// TwinCAT 3 PLC project bot53_plccode2
// ProgramVersion: 3.1.4022.7
// libraries:
//   CAA Memory, * (CAA Technical Workgroup)
//   Tc2_Math, * (Beckhoff Automation GmbH)
//   Tc2_SerialCom, * (Beckhoff Automation GmbH)
//   Tc2_Standard, * (Beckhoff Automation GmbH)
//   Tc2_System, * (Beckhoff Automation GmbH)
//   Tc2_Utilities, * (Beckhoff Automation GmbH)
//   Tc3_Database, * (Beckhoff Automation GmbH)
//   Tc3_IotBase, * (Beckhoff Automation GmbH)
//   Tc3_IotCommunicator, * (Beckhoff Automation GmbH)
//   Tc3_JsonXml, * (Beckhoff Automation GmbH)
//   Tc3_Module, * (Beckhoff Automation GmbH)
//   TcMatrix, * (Burks Engineering)
// project tree:
//   / CanRecTask.TcTTO, MqttTask.TcTTO, PlcTask.TcTTO
//   DUTs/ ST_IMU_STATE.TcDUT, ST_COMMAND.TcDUT, ST_FBDATA.TcDUT, ST_TARGETS.TcDUT, ST_UPCAM.TcDUT
//   GVLs/ GVL.TcGVL
//   POUs/ CanReceiver.TcPOU, constrain_angle.TcPOU, detectStabilizedAngle.TcPOU, DriveMotors.TcPOU, enable_disable_driver.TcPOU, FB_CanReceiver.TcPOU, FB_Mqtt.TcPOU, MAIN.TcPOU, motion_controller.TcPOU, MqttPrg.TcPOU, reset_errors.TcPOU, roundToTwoDecimalPlaces.TcPOU, set_encoder_odeometry.TcPOU, set_imu_odeometry.TcPOU, set_qr_info.TcPOU
//   POUs/kalman/ accum.TcPOU, angErrorCalc.TcPOU, angSpdCommandLimiter.TcPOU, angSpdCommandMixer.TcPOU, atan2.TcPOU, choldc1.TcPOU, choldcsl.TcPOU, cholsl.TcPOU, errorDegreeCalculator.TcPOU, forwardMovement.TcPOU, kalmanController.TcPOU, kalmanInit.TcPOU, kalmanStep.TcPOU, kinematicSolution.TcPOU, linPosErrGenerator.TcPOU, linSpdCommandLimiter.TcPOU, linSpdCommandMixer.TcPOU, localization.TcPOU, mulmat.TcPOU, myfmod.TcPOU, mySign.TcPOU, robotAutomation.TcPOU, setIdealAngle.TcPOU, ssub.TcPOU, sub_mat.TcPOU, transpose.TcPOU
// real-time tasks:
//   TASK CanRecTask: cycle T#2ms, priority 1, ADS port 350
//   TASK MqttTask: cycle T#10ms, priority 2, ADS port 351
//   TASK PlcTask: cycle T#2ms, priority 3, ADS port 352
// I/O:
//   DEVICE Device 3 (EtherCAT), AmsNetId 169.254.228.245.4.1
//     Term 1 (EK1960-2600) [EK1960-2600 TwinSAFE-Compact-Controller (4 x Relay, RJ45)]
//       modules: Module 1 (FSoE), Module 2 (FSOUT), Module 3 (FSLOGIC)
//       Term 2 (EL9410) [EL9410 E-Bus Power Supplier  (Diagnostics)]
//       Term 3 (EL3052) [EL3052 2Ch. Ana. Input 4-20mA]
//       Term 4 (EL2008-0015) [EL2008-0015 8Ch. Dig. Output 24V DC, 0.35A, not short-circuit proof]
//       Term 16 (EL9011) [EL9011 End Terminal]
//     Lifter_Driver [SOMANET CiA402 Drive]
//     Rotator_Driver [SOMANET CiA402 Drive]
//     Locomotion_R [SOMANET CiA402 Drive]
//     Locomotion_L [SOMANET CiA402 Drive]
//   DEVICE Device 1 (RT-Ethernet Adapter)
// variable links:
//   bot53_plccode2/bot53_plccode2 Instance <-> Device 3 (EtherCAT)/Lifter_Driver
//     MqttTask Inputs/GVL.robotdata.Position_Velocity.Lifter_position_actual_value <-> TxPDO Mapping 1/Position actual value
//     MqttTask Outputs/GVL.robotdata.Position_Velocity.Lifter_target_position <-> RxPDO Mapping 1/Target position
//     MqttTask Outputs/GVL.robotdata.motorCword[2] <-> RxPDO Mapping 1/Controlword
//     PlcTask Inputs/GVL.Lifter_modesOfOperationDisplay <-> TxPDO Mapping 1/Modes of operation display
//     PlcTask Inputs/GVL.Lifter_statusword <-> TxPDO Mapping 1/Statusword
//     PlcTask Inputs/GVL.batteryVoltageINT <-> TxPDO Mapping 1/batteryVoltage
//     PlcTask Inputs/GVL.robotdata.motorError[2] <-> TxPDO Mapping 1/Error code
//     PlcTask Outputs/GVL.Lifter_modesOfOperation <-> RxPDO Mapping 1/Modes of operation
//   bot53_plccode2/bot53_plccode2 Instance <-> Device 3 (EtherCAT)/Locomotion_L
//     MqttTask Outputs/GVL.robotdata.Position_Velocity.Locomotion_1_target_velocity <-> RxPDO Mapping 1/Target velocity
//     MqttTask Outputs/GVL.robotdata.motorCword[1] <-> RxPDO Mapping 1/Controlword
//     PlcTask Inputs/GVL.Locomotion_1_actual_pos <-> TxPDO Mapping 1/Position actual value
//     PlcTask Inputs/GVL.Locomotion_1_modesOfOperationDisplay <-> TxPDO Mapping 1/Modes of operation display
//     PlcTask Inputs/GVL.robotdata.Position_Velocity.Locomotion_1_actual_velocity <-> TxPDO Mapping 1/Velocity actual value
//     PlcTask Inputs/GVL.robotdata.motorError[1] <-> TxPDO Mapping 1/Error code
//     PlcTask Outputs/GVL.Locomotion_1_modesOfOperation <-> RxPDO Mapping 1/Modes of operation
//   bot53_plccode2/bot53_plccode2 Instance <-> Device 3 (EtherCAT)/Locomotion_R
//     MqttTask Outputs/GVL.robotdata.Position_Velocity.Locomotion_2_target_velocity <-> RxPDO Mapping 1/Target velocity
//     MqttTask Outputs/GVL.robotdata.motorCword[0] <-> RxPDO Mapping 1/Controlword
//     PlcTask Inputs/GVL.Locomotion_2_actual_pos <-> TxPDO Mapping 1/Position actual value
//     PlcTask Inputs/GVL.Locomotion_2_modesOfOperationDisplay <-> TxPDO Mapping 1/Modes of operation display
//     PlcTask Inputs/GVL.robotdata.Position_Velocity.Locomotion_2_actual_velocity <-> TxPDO Mapping 1/Velocity actual value
//     PlcTask Inputs/GVL.robotdata.motorError[0] <-> TxPDO Mapping 1/Error code
//     PlcTask Outputs/GVL.Locomotion_2_modesOfOperation <-> RxPDO Mapping 1/Modes of operation
//   bot53_plccode2/bot53_plccode2 Instance <-> Device 3 (EtherCAT)/Rotator_Driver
//     MqttTask Inputs/GVL.robotdata.Position_Velocity.Rotator_position_actual_value <-> TxPDO Mapping 1/Position actual value
//     MqttTask Outputs/GVL.robotdata.Position_Velocity.Rotator_target_position <-> RxPDO Mapping 1/Target position
//     MqttTask Outputs/GVL.robotdata.motorCword[3] <-> RxPDO Mapping 1/Controlword
//     PlcTask Inputs/GVL.Rotator_modesOfOperationDisplay <-> TxPDO Mapping 1/Modes of operation display
//     PlcTask Inputs/GVL.Rotator_statusword <-> TxPDO Mapping 1/Statusword
//     PlcTask Inputs/GVL.robotdata.motorError[3] <-> TxPDO Mapping 1/Error code
//     PlcTask Outputs/GVL.Rotator_modesOfOperation <-> RxPDO Mapping 1/Modes of operation
//   bot53_plccode2/bot53_plccode2 Instance <-> Device 3 (EtherCAT)/Term 1 (EK1960-2600)/Term 3 (EL3052)
//     PlcTask Inputs/GVL.robotdata.lifterDistance <-> AI Standard Channel 1/Value
//   bot53_plccode2/bot53_plccode2 Instance <-> Device 3 (EtherCAT)/Term 1 (EK1960-2600)/Term 4 (EL2008-0015)
//     MqttTask Outputs/GVL.robotdata.chargerContactor <-> Channel 3/Output
//     MqttTask Outputs/GVL.robotdata.driverContactor <-> Channel 1/Output
//     MqttTask Outputs/GVL.robotdata.pfEnableContactor <-> Channel 2/Output

CONFIGURATION bot53_plccode2
    RESOURCE PLC ON TwinCAT3
        TASK CanRecTask(INTERVAL := T#2ms, PRIORITY := 1);
        TASK MqttTask(INTERVAL := T#2ms, PRIORITY := 2);
        TASK PlcTask(INTERVAL := T#2ms, PRIORITY := 3);
        PROGRAM CanReceiver WITH CanRecTask : CanReceiver;
        PROGRAM MqttPrg WITH MqttTask : MqttPrg;
        PROGRAM robotAutomation WITH MqttTask : robotAutomation;
        PROGRAM MAIN WITH PlcTask : MAIN;
    END_RESOURCE
END_CONFIGURATION

// ---- DUTs/ST_IMU_STATE.TcDUT
TYPE ST_IMU_STATE :
STRUCT
	imu_x:LREAL;
	imu_y:LREAL;
	imu_euler:LREAL;
	acc_x:LREAL;
	gyro_z:LREAL;
	hr_acc_x:LREAL;
	hr_gyro_z:LREAL;
	timediff:LREAL;
	euler_yaw:LREAL;
END_STRUCT
END_TYPE

// ---- DUTs/ST_COMMAND.TcDUT
TYPE ST_COMMAND :
STRUCT
	command:INT;
	distance:LREAL;
	direction:INT;
	acc:LREAL;
	jerk:LREAL;
	spd:LREAL;
END_STRUCT
END_TYPE

// ---- DUTs/ST_FBDATA.TcDUT

TYPE ST_FBDATA :
STRUCT
    robot_x:LREAL;
	robot_y:LREAL;
	robot_yaw:LREAL;
	lifter:LREAL;
	rotator:LREAL;
	upcam_state:st_upcam;
	batteryStatus:BYTE;
	batteryVoltage :LREAL := 50;
	batteryRequestCurrent:LREAL;
	batterySOC:INT:=90;
	batteryCurrentCons:LREAL;
	batteryErrorFlag:INT;
	qr_tag:INT:=0;
	qr_x:INT;
	qr_y:INT;
	qr_angle:INT;
	qr_yaw:LREAL:=0;
	imu_state:ST_IMU_STATE;
	deviation_yaw:LREAL;
	deviation_y:LREAL;
	imu_r:LREAL;
	imu_omega:LREAL;
	imu_readtime:LREAL;
	encoder_x:LREAL;
	encoder_y:LREAL;
	encoder_yaw:LREAL;
	encoder_v:LREAL;
	robot_direction:BYTE:=0;
	motion_status :BYTE:=1;
	activeState:BYTE:=1;
	
	motorError AT%I*:ARRAY[0..3] OF INT;
	Jerk:LREAL:=JERK_LIMIT;
	Acc:LREAL:=ACCELERATION_LIMIT;
	Speed:LREAL:=SPEED_LIMIT;
	controller:INT;
	motorCword AT%Q*: ARRAY[0..3] OF INT;
	yaw_error:LREAL;
	encoder_omega:LREAL;
	encoder_slave0_speed:LREAL;
	encoder_slave1_speed:LREAL;
	encoderx_rel:LREAL;
	encodery_rel:LREAL;
	imux_rel:LREAL;
	imuy_rel:LREAL;
	wc1:LREAL;
	wc2:LREAL;
	driverContactor                            AT%Q* : BOOL := TRUE;
    pfEnableContactor                        AT%Q* : BOOL := TRUE;
    chargerContactor                        AT%Q* : BOOL := FALSE;
	lifterDistance AT%I* : INT := INT#0;
	Position_Velocity:ST_TARGETS;
	activecommand:INT;
	Locomotion_1_modesOfOperationDisplay    AT%I* : SINT;
	Locomotion_2_modesOfOperationDisplay    AT%I* : SINT;
    Rotator_modesOfOperationDisplay         AT%I* : SINT;
    Lifter_modesOfOperationDisplay          AT%I* : SINT;
  
	END_STRUCT
	END_TYPE

// ---- DUTs/ST_TARGETS.TcDUT
TYPE ST_TARGETS :
STRUCT
	Locomotion_1_target_velocity			AT%Q* : DINT;
	Locomotion_2_target_velocity 			AT%Q* : DINT;
	Locomotion_1_actual_velocity			AT%I* : DINT;
	Locomotion_2_actual_velocity 			AT%I* : DINT;
	Lifter_position_actual_value             AT%I* : DINT;
	Lifter_target_position                     AT%Q* : DINT;
	Rotator_target_position                 AT%Q* : DINT;
	Rotator_position_actual_value             AT%I* : DINT;
	Rotator_target_velocity                 AT%Q* : DINT;
	Rotator_actual_velocity             AT%I* : DINT;
END_STRUCT
END_TYPE

// ---- DUTs/ST_UPCAM.TcDUT
TYPE ST_UPCAM :
STRUCT
	up_camera_x:LREAL;
	up_camera_y:LREAL;
	up_camera_yaw:LREAL;
	up_camera_tag:STRING[10];
END_STRUCT
END_TYPE

// ---- GVLs/GVL.TcGVL
//{attribute 'qualified_only'}
VAR_GLOBAL CONSTANT
COMMAND_LOCOMOTION_DISABLE:BYTE:=BYTE#2;
COMMAND_LOCOMOTION_ENABLE:BYTE:=BYTE#14;
COMMAND_LIFTER_DISABLE:BYTE:=BYTE#6;
COMMAND_LIFTER_ENABLE:BYTE:=BYTE#7;
COMMAND_ROTATOR_DISABLE:BYTE:=BYTE#8;
COMMAND_ROTATOR_ENABLE:BYTE:=BYTE#9;
COMMAND_PF_ENADIS:BYTE:=BYTE#11;
COMMAND_DRIVER_ENADIS:BYTE:=BYTE#12;
COMMAND_RESET_ERRORS:BYTE:=BYTE#1;
COMMAND_SET_MOTIONLIMITS:BYTE:=BYTE#21;
COMMAND_TOGGLE_CONT:BYTE:=BYTE#33;
COMMAND_CANCEL_COMMAND:BYTE:=BYTE#36;
COMMAND_ANG_CORR:BYTE:=BYTE#32;
COMMAND_X_CORR:BYTE:=BYTE#34;
MOTION_ONGOING:BYTE:=BYTE#0;
GRID_DIM:INT:=INT#1;
//QR_TX_INTERVAL:LREAL:=LREAL#25;
MOTION_ENDED:BYTE:=BYTE#1;
MOTION_INFINITE:BYTE:=BYTE#2;
MOTION_HOLDED:BYTE:=BYTE#3;
MOTION_ANGLE:BYTE:=BYTE#4;
MOTION_LIFTER:BYTE:=BYTE#5;
STARTSTOP_CHARGE:BYTE:=BYTE#45;
MOTION_OBSTACLE:BYTE:=BYTE#7;
MOTION_ROTATE:BYTE:=BYTE#8;
CHARGING:BYTE:=BYTE#9;
LIFTER_UP_LIMIT:INT:=INT#14879;
LIFTER_DOWN_LIMIT:INT:=INT#32000;
LIFTER_UP:INT:=INT#16000;
LIFTER_DOWN:INT:=INT#25000;

MOTION_BRAKE:BYTE:=BYTE#10;
IMU_RESET :BYTE:=BYTE#11;
ANGLE_CORRECT:BYTE:=BYTE#12;
LOCATION_CORRECT:BYTE:=BYTE#13;
INIT:BYTE:=BYTE#14;
LIFTING_DONE:BYTE:=BYTE#15;
POD_ANGLE_CORRECT:BYTE:=BYTE#16;
ENC_RESET :BYTE:=BYTE#17;
PDO_CHARGE_OPENCLOSE:BYTE:=BYTE#18;
STOP_ON_QR :BYTE:=BYTE#19;
UPCAM_READ:BYTE:=BYTE#20;
ANGLE_CORR_ENDED :BYTE:=BYTE#50;
X_CORR_ENDED :BYTE:=BYTE#51;
POD_CORR_ENDED:BYTE:=BYTE#52;
IMU_RST_ENDED:BYTE:=BYTE#53;
CONT_TOGGLE_ENDED :BYTE:=BYTE#54;
MOVE_ENDED :BYTE:=BYTE#55;
TURN_ENDED :BYTE:=BYTE#56;
LIFT_ENDED :BYTE:=BYTE#57;
ROTATE_ENDED :BYTE:=BYTE#58;
SETLIMITS_ENDED :BYTE:=BYTE#59;
CHARGE_ENDED:BYTE:=BYTE#60;
UPCAM_READ_ENDED :BYTE:=BYTE#61;
LIFT_UP:BYTE:=BYTE#62;
LIFT_DOWN:BYTE:=BYTE#63;
LOST:BYTE:=BYTE#100;
MOTOR_ERROR:BYTE:=BYTE#105;
PLC_ERROR:BYTE:=BYTE#106;
IMU_ERROR:BYTE:=BYTE#107;
NO_QR_TIMEOUT:DINT:=DINT#50000000;
NO_ADS_TIMEOUT:DINT:=DINT#150;
QRCAM_ERROR:BYTE:=BYTE#110;
COMM_PROB:BYTE:=BYTE#111;
CMD_TIMEOUT :BYTE:=BYTE#112;
STOPPER_DOWN:BYTE:=BYTE#114;
UPCAM_ERROR:BYTE:=BYTE#115; //error states starting from 100
PLC_COMM_ERROR :BYTE:=BYTE#116;
BMS_ERROR:BYTE:=BYTE#120;
PDO_CHARGER_ERROR :BYTE:=BYTE#121;
CRI_BATT:BYTE:=BYTE#125;
OVER_CURR:BYTE:=BYTE#126;
CHARGE_ERROR:BYTE:=BYTE#127;
LOW_BATT:BYTE:=BYTE#130;
MOTOR_OVER_TEMP:BYTE:=BYTE#135;
BATT_ERROR:BYTE:=BYTE#150;
LIFTER_STATE_INCORRECT:BYTE:=BYTE#160;

 

SUCCESS:INT:=INT#0;
FAILURE:INT:=INT#2;
NEGATIVE_FAILURE:INT:=INT#3;
NULL_POINTER:INT:=INT#4;
ROBOT_RADIUS:LREAL:=LREAL#0.32;
WHEEL_RADIUS:LREAL:=LREAL#0.08;
REDUCER_RATIO:LREAL:=LREAL#12;
ROTATOR_RADIUS:LREAL:=LREAL#0.466;
TURN_JERK_LIMIT:LREAL:=LREAL#0.4;
TURN_ACCELERATION_LIMIT:LREAL:=LREAL#0.2;
TURN_VELOCITY_LIMIT:LREAL:=LREAL#0.2;


DECELERATION_LIMIT:LREAL:=LREAL#1;

PLC_CYCLE:LREAL:=LREAL#0.002;
ROTATOR_REDUCER_RATIO:LREAL:=LREAL#14;
ROTATOR_GEAR_RATIO:LREAL:=LREAL#7.6;
ROTRAD2DEC:LREAL:=(10000.0 * (ROTATOR_REDUCER_RATIO) * (ROTATOR_GEAR_RATIO) / (2.0 * PI));
DEC2R:LREAL:=LREAL#1/ROTRAD2DEC;
M2DEC:LREAL:=((10000.0 * (REDUCER_RATIO)) / (2.0 * PI * (WHEEL_RADIUS)));
DEC2M:LREAL:= (1.0 / (M2DEC));
MSN2RPM:LREAL:= ((((REDUCER_RATIO) * 1.0 * 60.0) / (2.0 * PI * (WHEEL_RADIUS))));
RPM2MSN:LREAL:=1/MSN2RPM;
OMEGA_DIFF_MAX:LREAL:= ((1.5 * 1.5) / (ROBOT_RADIUS * ROBOT_RADIUS) * (PLC_CYCLE));

END_VAR
VAR_GLOBAL
imu_euler_prev:LREAL;
qr_xstate:LREAL;
qr_ystate:LREAL;
slave0_speed:LREAL;
slave1_speed:LREAL;
ACCELERATION_LIMIT:LREAL:=LREAL#1;
JERK_LIMIT:LREAL:=LREAL#0.8;
SPEED_LIMIT:LREAL:=LREAL#1.5;
//******************KALMAN VARIABLES**********************************************
	LINSPDRATELIMIT:LREAL:= 0.7;
	LINPOS_Kp :LREAL:=0.85;
	TURNANG_Kp:LREAL:= 1.5;
	TURNFWD_Kp:LREAL:= 1.5;
	FORWARD_MAX_SPEED :LREAL:=1.5;
	LINJERKLIMIT:LREAL:= 20;
	ANGSPDRATELIMIT :INT:= 20;
	calibrationCount:INT:=0;
	gyroZmean:LREAL:=0;
	accXmean:LREAL:=0; 
	PosFdbckX,PosFdbckX_Rel:LREAL:=0;
	PosFdbckY,PosFdbckY_Rel:LREAL:=0;
	ThetaFdbck:LREAL:=0;
	xStart:LREAL:=0;
	yStart:LREAL:=0;
	xGoal:LREAL:=0;
	yGoal:LREAL:=0;
	idealAngle:LREAL:=0;
	AngPosCommand:LREAL:=0;
	robotAngle:LREAL:=0;
	linPosErr:LREAL:=0;
	kalLinSpd:LREAL:=0;
	kalAngSpd:LREAL:=0;
	linSpdCommandShaped:LREAL:=0;angSpdCommandShaped:LREAL:=0;angPosFdbckRobot_Abs:LREAL:=0;angPosFdbckRobot:LREAL:=0; angSpdFdbckRobot_:LREAL:=0; linPosFdbckRobot_x:LREAL:=0; linSpdFdbckRobot_x_:LREAL:=0;linSpdFdbckRobot:LREAL:=0;
	angSpdFdbckRobot:LREAL:=0; linPosFdbckRobot_y:LREAL:=0; linSpdFdbckRobot_y_:LREAL:=0;rightWheelFdbck:LREAL:=0;leftWheelFdbck:LREAL:=0;
	robot_state:BYTE:=0;modeEnable:BYTE:=0;missionCompleted:INT:=1;userCommand:BYTE:=0; readyFlag:BYTE:=0;
	rightMotorSpeedCommand:DINT;leftMotorSpeedCommand:DINT;
	posTheta_wrt_robot_enc:LREAL;
	forwardCommand:LREAL:= 0;
	accLimited :LREAL:= 0;
	LinSpdFdbck:LREAL:=0;accFdbck:LREAL:=0;linSpd:LREAL:=0;
	Id:DynamicMatrix;
	I:ARRAY[0..2,0..2] OF LREAL:=[1,0,0,0,1,0,0,0,1];
	F_kalman1:ARRAY[0..2,0..2] OF LREAL:=[1,0.002,0.000002,0,1,0.002,0,0,1];	
	Q_kalman1:ARRAY[0..2,0..2] OF LREAL:=[0,0,0,0,0,0,0,0,10];
	R_kalman1:ARRAY[0..1,0..1] OF LREAL:=[1,0,0,1000];
	x_kalman1:ARRAY[0..2,0..0] OF LREAL:=[0,0,0];
	P_kalman1:ARRAY[0..2,0..2]OF LREAL:=[1,0,0,0,1,0,0,0,1];
	z_kalman1:ARRAY[0..1,0..0] OF LREAL;
	K_kalman1:ARRAY[0..2,0..1]OF LREAL;
	H_kalman1:ARRAY[0..1,0..2] OF LREAL:=[1,0,0,0,1,0];
	F_kalman2:ARRAY[0..2,0..2] OF LREAL:=[1,0.002,0.000002,0,1,0.002,0,0,1];
	Q_kalman2:ARRAY[0..2,0..2] OF LREAL:=[0,0,0,0,0,0,0,0,10];
	R_kalman2:ARRAY[0..1,0..1] OF LREAL:=[1,0,0,1];
	x_kalman2:ARRAY[0..2,0..0] OF LREAL:=[0,0,0];
	P_kalman2:ARRAY[0..2,0..2] OF LREAL:=[1,0,0,0,1,0,0,0,10];
	z_kalman2:ARRAY[0..1,0..0] OF LREAL;
	K_kalman2:ARRAY[0..2,0..1]  OF LREAL;
	H_kalman2:ARRAY[0..1,0..2] OF LREAL:=[1,0,0,0,1,0];
	err_kalman2:ARRAY[0..1,0..0] OF LREAL;
	F_kalman3:ARRAY[0..2,0..2] OF LREAL:=[1,0,0,0,1,0,0,0,1];
	Q_kalman3:ARRAY[0..2,0..2]  OF LREAL:=[10,0,0,0,10,0,0,0,0.2];
	R_kalman3:ARRAY[0..2,0..2] OF LREAL:=[0.01,0,0,0,0.01,0,0,0,500]; 
	x_kalman3:ARRAY[0..2,0..0]OF LREAL:=[0,0,0];
	z_kalman3:ARRAY[0..2,0..0]OF LREAL:=[0,0,0];
	P_kalman3:ARRAY[0..2,0..2]OF  LREAL:=[1,0,0,0,1,0,0,0,1];
	H_kalman3:ARRAY[0..2,0..2] OF LREAL;
	K_kalman3:ARRAY[0..2,0..2]OF LREAL;
	theta_pos:LREAL := 0;
	kalman12_x:LREAL;
	kalman12_y :LREAL;
	err_kalman3:ARRAY[0..2,0..0]OF LREAL;

//******************KALMAN VARIABLES**********************************************

	CONTROLLER_TYPE:BYTE:=0;
	KALMAN_INITIALIZED:BOOL:=FALSE;
	Y_DEV_THRESHOLD:LREAL:=0.005;
	PF_OFFSET:LREAL:=-0.4;
	pf_valid:BYTE:=0;
	AWAY_COEFF:LREAL:=LREAL#1;
	TOWARDS_COEFF:LREAL:=LREAL#1;
    current_yaw_deg:LREAL;
    ads_lasttime:ULINT;
    lateral_direction_sign:INT;
	batteryVoltageINT  AT%I*:UDINT;
    away:LREAL;
	cancelcommand:BOOL;
	raw_qr_tag:INT;
      stabilization_yaw_deg:LREAL;
    winnerEvaluated:BOOL:=FALSE;
    imuXwins:BOOL:=FALSE;
	imuAngwins:BOOL:=FALSE;
    lastqrtime:ULINT;
	lastqrtagtime:ULINT;
    controller_coeff:LREAL;
    imuYwins:BOOL:=FALSE;
    encoderx_rel:LREAL;
    encodery_rel:LREAL;
    imux_rel:LREAL;
    imuy_rel:LREAL;
	grid_x:LREAL;
	grid_y:LREAL;
    local_x_before_motion:LREAL:=0;
     robotdata:ST_FBDATA;
    st_command:ST_COMMAND;
    command:ARRAY[0..5] OF LREAL;
    motion_index :DINT;
    max_location :DINT;
    motion_left  :ARRAY[0..299999] OF DINT;
	motion_lift  :ARRAY[0..299999] OF DINT;
	motion_rotator  :ARRAY[0..299999] OF DINT;
    motion_right :ARRAY[0..299999] OF DINT;
    motion_vel :ARRAY[0..299999] OF LREAL;
    motion  :ARRAY[0..299999] OF DINT;
    deviation_y:LREAL;
    deviation_yaw:LREAL;
    KpY:LREAL:=95;
    KpTht:LREAL:=0.03;
    //Locomotion_1
    Locomotion_1_modesOfOperation             AT%Q* : SINT := SINT#9;
    Locomotion_1_error_state_1                 AT%I* : UINT;
    Locomotion_1_error_state_2                 AT%I* : UINT;
    Locomotion_1_statusword                 AT%I* : UINT;
	Locomotion_1_actual_pos                 AT%I* : DINT;
    Locomotion_1_modesOfOperationDisplay     AT%I* : SINT;
    //Locomotion_2

    Locomotion_2_modesOfOperation             AT%Q* : SINT := SINT#9;
    Locomotion_2_error_state_1                 AT%I* : UINT;
    Locomotion_2_error_state_2                 AT%I* : UINT;
    Locomotion_2_statusword                 AT%I* : UINT;
    Locomotion_2_modesOfOperationDisplay     AT%I* : SINT;
	Locomotion_2_actual_pos                 AT%I* : DINT;
    //Rotator
   
    Rotator_modesOfOperation                 AT%Q* : SINT := SINT#8;
  
    Rotator_error_state_1                     AT%I* : UINT;
    Rotator_error_state_2                     AT%I* : UINT;
    Rotator_statusword                         AT%I* : UINT;
    Rotator_modesOfOperationDisplay         AT%I* : SINT;
    //Lifter
  
    Lifter_modesOfOperation                 AT%Q* : SINT := SINT#8;
   
    Lifter_error_state_1                     AT%I* : UINT;
    Lifter_error_state_2                     AT%I* : UINT;
    Lifter_statusword                         AT%I* : UINT;
    Lifter_modesOfOperationDisplay             AT%I* : SINT;
    receivedBytes :STRING;
    sendReceiveTrigger : BOOL;

    MQTT_ConnState:ETcIotMqttClientState;
    MQTT_Command:FB_IoTCommand;

    //Enable Signals for to be switched subsystems
   

 


END_VAR

// ---- POUs/CanReceiver.TcPOU
PROGRAM CanReceiver
VAR
	fbUdp1 : FB_CanReceiver;
END_VAR

fbUdp1();

END_PROGRAM

// ---- POUs/FB_CanReceiver.TcPOU
{attribute 'c++_compatible'}
FUNCTION_BLOCK FB_CanReceiver IMPLEMENTS ITcIoUdpProtocolRecv
VAR_INPUT
END_VAR
VAR_OUTPUT
END_VAR
VAR
	{attribute 'TcInitSymbol'}
	oid : OTCID; 
	ipUdp : ITcIoUdpProtocol;
	nUdpPort : UINT := 4444;
	nReceivedPakets : UINT;
	
	hrInit : HRESULT;
	hrSend  : HRESULT;  
END_VAR

IF ipUdp <> 0 THEN
	ipUdp.CheckReceived();
END_IF

{attribute 'conditionalshow'}
METHOD FB_exit : BOOL
VAR_INPUT
	bInCopyCode : BOOL; // if TRUE, the exit method is called for exiting an instance that is copied afterwards (online change).
END_VAR
IF NOT bInCopyCode THEN // no online change
	IF ipUdp <> 0 THEN 
		ipUdp.UnregisterReceiver(nUdpPort); // Shutdown
		FW_SafeRelease(ADR(ipUdp));
		FB_exit := TRUE; 
	END_IF
END_IF
END_METHOD

{attribute 'conditionalshow'}
METHOD FB_init : BOOL
VAR_INPUT
	bInitRetains : BOOL; // if TRUE, the retain variables are initialized (warm start / cold start)
	bInCopyCode : BOOL;  // if TRUE, the instance afterwards gets moved into the copy code (online change)
END_VAR
VAR
	ipSrv : ITComObjectServer;

END_VAR
IF NOT bInCopyCode THEN // no online change
	IF ipUdp = 0 AND oid <> 0 THEN
	    hrInit := FW_ObjMgr_GetObjectInstance(	oid:=oid, 
											iid:=TC_GLOBAL_IID_LIST.IID_ITcIoUdpProtocol, 
											pipUnk:=ADR(ipUdp) );
		IF SUCCEEDED(hrInit) THEN 
			IF  SUCCEEDED(ipUdp.RegisterReceiver(nUdpPort, THIS^)) THEN //open port
				FB_init := TRUE;
			ELSE 
				FB_init := FALSE; 
				FW_SafeRelease(ADR(ipUdp));
			END_IF
		END_IF
	ELSIF oid = 0 THEN 
		FB_init := FALSE; 
		hrInit := ERR_INVALID_PARAM; 				
	END_IF
END_IF
END_METHOD

{attribute 'conditionalshow'}
METHOD FB_reinit : BOOL
VAR_INPUT
END_VAR
IF (ipUdp <> 0) THEN 
	ipUdp.RegisterReceiver(nUdpPort, THIS^);
	FB_reinit := TRUE; 
END_IF
END_METHOD

{attribute 'object_name' := 'ReceiveData'}
{attribute 'c++_compatible'}
{attribute 'signature_flag' := '33554688'}
{attribute 'pack_mode' := '4'}
{attribute 'show'}
{attribute 'minimal_input_size' := '4'}
METHOD ReceiveData : HRESULT
VAR_INPUT
	ipAddr	: UDINT;
	udpDestPort	: UINT;
	udpSrcPort	: UINT;
	nData	: UDINT;
	pData	: PVOID;
	pVlan	: POINTER TO ETYPE_VLAN_HEADER := 0;
END_VAR
VAR
	receivedBytes:ARRAY[0..9]OF BYTE;
	fbTime:FB_LocalSystemTime;
	 tStruct: TIMESTRUCT;
	  msec: DINT;
	  datatype:BYTE;
    dTime: DATE_AND_TIME;
    eTime_sec: DINT;
	FB_QR:set_qr_info();
    eTime_msec: LINT;
END_VAR


IF ipUdp <> 0 THEN
	
	MEMCPY( ADR(robotdata.qr_x), pData, 2 );
	MEMCPY( ADR(robotdata.qr_y), pData+2, 2 );
	MEMCPY( ADR(robotdata.qr_angle), pData+4, 2 );
	MEMCPY( ADR(raw_qr_tag), pData+6, 2 );
	MEMCPY( ADR(pf_valid), pData+8, 1 );
	fbTime(bEnable:=TRUE, dwCycle:=1, SystemTime=>tStruct);
	msec := tStruct.wMilliseconds;
	tStruct.wMilliseconds := 0;
	dTime := SYSTEMTIME_TO_DT(tStruct);
	eTime_sec := DT_TO_DINT(dTime);
	lastQrtime := F_GetSystemTime() ;	
	FB_QR();
//LAST QR TIME ALINACAK
	
END_IF
END_METHOD

{attribute 'object_name' := 'TcAddRef'}
{attribute 'c++_compatible'}
{attribute 'signature_flag' := '33554688'}
{attribute 'pack_mode' := '4'}
{attribute 'show'}
{attribute 'minimal_input_size' := '4'}
METHOD TcAddRef : UDINT
END_METHOD

{attribute 'object_name' := 'TcQueryInterface'}
{attribute 'c++_compatible'}
{attribute 'signature_flag' := '33554688'}
{attribute 'pack_mode' := '4'}
{attribute 'show'}
{attribute 'minimal_input_size' := '4'}
METHOD TcQueryInterface : HRESULT
VAR_INPUT
	iid	: REFERENCE TO IID;
	pipItf	: POINTER TO PVOID;
END_VAR
VAR
	ipUdpRecv : ITcIoUdpProtocolRecv;
	ipUnknown : ITcUnknown;	
END_VAR
IF GuidsEqual(ADR(iid), ADR(TC_GLOBAL_IID_LIST.IID_ITcIoUdpProtocolRecv)) THEN
	ipUdpRecv := THIS^; // cast to interface pointer
	pipItf^ := ITCUNKNOWN_TO_PVOID(ipUdpRecv);
	TcAddRef();
	TcQueryInterface := S_OK;
ELSIF GuidsEqual(ADR(iid), ADR(TC_GLOBAL_IID_LIST.IID_ITcUnknown)) THEN
	ipUnknown := THIS^; // cast to interface pointer
	pipItf^ := ITCUNKNOWN_TO_PVOID(ipUnknown);
	TcAddRef();
	TcQueryInterface := S_OK;
ELSE
	TcQueryInterface := E_HRESULTAdsErr.NOINTERFACE ; //Call super if this fb extends some other
END_IF
END_METHOD

{attribute 'object_name' := 'TcRelease'}
{attribute 'c++_compatible'}
{attribute 'signature_flag' := '33554688'}
{attribute 'pack_mode' := '4'}
{attribute 'show'}
{attribute 'minimal_input_size' := '4'}
METHOD TcRelease : UDINT
END_METHOD

END_FUNCTION_BLOCK

// ---- POUs/set_qr_info.TcPOU
FUNCTION_BLOCK PUBLIC set_qr_info

VAR
	modified_qr:DINT;
	
END_VAR

   IF(pf_valid=1) THEN 
	lastqrtagtime := F_GetSystemTime() ;
 // END_IF	
 // IF(raw_qr_tag<>0 AND ((robotdata.robot_direction MOD 2 =0 AND robotdata.qr_x<>0) OR (robotdata.robot_direction MOD 2 =1 AND robotdata.qr_y<>0))) THEN
  	modified_qr:=raw_qr_tag;
    IF(raw_qr_tag>=82 AND raw_qr_tag<102)  THEN
      robotdata.qr_tag := raw_qr_tag-61;
      grid_x := (robotdata.qr_tag-1)/5;
      grid_y := (robotdata.qr_tag-1) MOD 5;
    
    ELSIF(raw_qr_tag>101)THEN
      modified_qr := raw_qr_tag-102;
      robotdata.qr_tag := raw_qr_tag-61;
      grid_x := (modified_qr)/4;
      grid_y := (modified_qr) MOD 4+5;
    ELSIF(raw_qr_tag>40)THEN
      grid_x := (robotdata.qr_tag-41)/4;
      grid_y := (robotdata.qr_tag-41) MOD 4+5;
     robotdata.qr_tag :=raw_qr_tag;
    ELSE
	grid_x := (robotdata.qr_tag-1)/5;
    grid_y := (robotdata.qr_tag-1) MOD 5;
	robotdata.qr_tag :=raw_qr_tag;
	END_IF
    robotdata.qr_yaw :=  LMOD((-robotdata.qr_angle * 0.1-PF_OFFSET) * PI / 180.0+(2*PI) , (2*PI));
    robotdata.robot_x := (grid_x * GRID_DIM) + (robotdata.qr_x / 1000.0) + (robotdata.encoder_v * COS(robotdata.qr_yaw) * PLC_CYCLE ); //the constant at the end is based on the latency of the camera
    robotdata.robot_yaw:=robotdata.qr_yaw;
    IF(  NOT winnerEvaluated AND ABS(LMOD(robotdata.imu_state.imu_euler + 2*PI,2*PI)- robotdata.qr_yaw)<ABS(LMOD(robotdata.encoder_yaw + 2*PI,2*PI)-robotdata.qr_yaw)) THEN
      imuAngwins:=TRUE;
    ELSIF( NOT winnerEvaluated AND  ABS(LMOD(robotdata.imu_state.imu_euler + 2*PI,2*PI)- robotdata.qr_yaw)>ABS(LMOD(robotdata.encoder_yaw + 2*PI,2*PI)-robotdata.qr_yaw)) THEN
      imuAngwins:=FALSE;
    END_IF
	  
    IF(  NOT winnerEvaluated AND ABS(robotdata.imux_rel-(robotdata.qr_x / 1000.0))<ABS(robotdata.encoderx_rel-(robotdata.qr_x / 1000.0))) THEN
      imuXwins:=TRUE;
    ELSIF( NOT winnerEvaluated AND ABS(robotdata.imux_rel-(robotdata.qr_x / 1000.0))>ABS(robotdata.encoderx_rel-(robotdata.qr_x / 1000.0))) THEN
      imuXwins:=FALSE;
	  END_IF
    
    robotdata.encoder_x := robotdata.robot_x;
    robotdata.imu_state.imu_x := robotdata.robot_x;
	
  
  
    robotdata.robot_y := (grid_y * GRID_DIM) + (robotdata.qr_y / 1000.0) + (robotdata.encoder_v * SIN(robotdata.qr_yaw) * PLC_CYCLE);
   IF( NOT winnerEvaluated AND  ABS(robotdata.imuy_rel-(robotdata.qr_y / 1000.0))<ABS(robotdata.encodery_rel-(robotdata.qr_y / 1000.0))) THEN
      imuYwins:=TRUE;
    ELSIF( NOT winnerEvaluated AND  ABS(robotdata.imuy_rel-(robotdata.qr_y / 1000.0))>ABS(robotdata.encodery_rel-(robotdata.qr_y / 1000.0))) THEN
      imuYwins:=FALSE;
	END_IF      
  
    winnerEvaluated:=TRUE;

   //printf("%d-%d\n",imuXwins,imuYwins);
    robotdata.encoder_y := robotdata.robot_y;
    robotdata.imu_state.imu_y :=robotdata.robot_y;
	//robotdata.imu_state.imu_euler:=robotdata.robot_yaw;
	robotdata.encoder_yaw:=robotdata.robot_yaw;
	//robotdata.encoder_yaw:=robotdata.qr_yaw;
    //imu_odometry->imu_euler=qr_info->yaw_state;
	qr_xstate:=robotdata.robot_x;
	qr_ystate:=robotdata.robot_y;
   ELSE
    winnerEvaluated:=FALSE;
	robotdata.qr_tag :=0;
	END_IF

END_FUNCTION_BLOCK

// ---- POUs/MqttPrg.TcPOU
PROGRAM MqttPrg
VAR
	fbMqttClient  : FB_Mqtt;
    bSetParameter : BOOL := TRUE;
	bHostnameSet:BOOL:=FALSE;
    bConnect      : BOOL := TRUE;
	bSubscribed : BOOL;
    sPayloadPub : STRING(2500);
	fbJson         : FB_JsonSaxWriter;
  	fbJsonDataType : FB_JsonReadWriteDataType;
	i: UDINT;
    fbTimer : TON := (PT:=T#10MS);
	hostnameexecuter:TON;
	gethostname:FB_GetHostName:=(sNetID:='',bExecute:=bHostnameSet);

	
END_VAR

IF(HOSTNAME='') THEN
hostnameexecuter(IN:=TRUE,PT:=T#1S,Q=>bHostnameSet);
gethostname(sNetID:='',bExecute:=bHostnameSet,sHostName=>HOSTNAME);
END_IF
IF  HOSTNAME<>'' AND bSetParameter  AND NOT fbMqttClient.bConnected THEN
    bSetParameter              := FALSE;
    fbMqttClient.sHostName     := '192.168.8.80';
    fbMqttClient.nHostPort     := 1883;
    fbMqttClient.sClientId     := HOSTNAME; 
    fbMqttClient.sTopicPrefix  := ''; 
	MQTT_FEEDBACK_TOPIC:=concat('FBDATA/',HOSTNAME);
	MQTT_COMMAND_TOPIC:=concat('COMMAND/',HOSTNAME);
//  fbMqttClient.nKeepAlive    := 60; 
//  fbMqttClient.sUserName     := ;
//  fbMqttClient.sUserPassword := ; 
//  fbMqttClient.stWill        := ; 
//  fbMqttClient.stTLS         := ;
	 
END_IF
IF(HOSTNAME<>'') THEN
	fbMqttClient.Execute(bConnect);
END_IF
IF fbMqttClient.bConnected THEN
    IF NOT bSubscribed THEN
        bSubscribed := fbMqttClient.Subscribe(sTopic:=MQTT_COMMAND_TOPIC, eQoS:=TcIotMqttQos.ExactlyOnceDelivery) AND fbMqttClient.Subscribe(sTopic:='STOPPER', eQoS:=TcIotMqttQos.ExactlyOnceDelivery);
    END_IF
    fbTimer(IN:=TRUE);
    IF fbTimer.Q THEN // publish new payload every second
        fbTimer(IN:=FALSE);
      	fbJson.ResetDocument();
		fbJsonDataType.AddJsonValueFromSymbol(fbJson, 'ST_FBDATA', SIZEOF(robotdata), ADR(robotdata));
		sPayloadPub := fbJson.GetDocument();
		fbJson.CopyDocument(sPayloadPub, SIZEOF(sPayloadPub));
        fbMqttClient.Publish(   sTopic:= MQTT_FEEDBACK_TOPIC, 
                                pPayload:= ADR(sPayloadPub), nPayloadSize:= LEN2(ADR(sPayloadPub))+1, 
                                eQoS:= TcIotMqttQos.AtMostOnceDelivery, bRetain:= FALSE, bQueue:= FALSE );
    END_IF
END_IF

END_PROGRAM

// ---- POUs/FB_Mqtt.TcPOU
{attribute 'c++_compatible'}
FUNCTION_BLOCK PUBLIC FB_Mqtt EXTENDS FB_IotMqttClient
VAR
    (* received message *)
    {attribute 'TcEncoding':='UTF-8'}
    sTopicRcv   : STRING(255);
    {attribute 'TcEncoding':='UTF-8'}
    sPayloadRcv : STRING(255);
END_VAR

{attribute 'c++_compatible'}
{attribute 'pack_mode' := '4'}
{attribute 'show'}
{attribute 'minimal_input_size' := '4'}
METHOD OnMqttMessage : HRESULT
VAR_IN_OUT CONSTANT
    topic    : STRING;
END_VAR
VAR_INPUT
    payload  : PVOID;
    length   : UDINT;
    qos      : TcIotMqttQos;
    repeated : BOOL;
END_VAR
VAR
    nPayloadRcvLen : UDINT;
	fbJsonDataType : FB_JsonReadWriteDataType;
	fbreseterrors:reset_errors;
	fbenadisloco:enable_disable_driver;
END_VAR

STRNCPY( ADR(sTopicRcv), ADR(topic), SIZEOF(sTopicRcv) );
nPayloadRcvLen := MIN(length, DINT_TO_UDINT(SIZEOF(sPayloadRcv))-1);
MEMCPY( ADR(sPayloadRcv), payload, nPayloadRcvLen );
sPayloadRcv[nPayloadRcvLen] := 0;  // ensure a null termination of received string
IF(topic=MQTT_COMMAND_TOPIC AND fbJsonDataType.SetSymbolFromJson(sPayloadRcv, 'ST_COMMAND', SIZEOF(st_command), ADR(st_command)))THEN
	robotdata.activecommand:=st_command.command;
	CASE st_command.command OF
	COMMAND_STOP:
		robotdata.motorCword[0]:=43;
		robotdata.motorCword[1]:=43;
	COMMAND_LOCOMOTION_DISABLE:
		fbenadisloco(DRIVER:=0,CWORD:=6);
	COMMAND_LOCOMOTION_ENABLE:
		fbenadisloco(DRIVER:=0,CWORD:=47);
	COMMAND_LIFTER_DISABLE:
		fbenadisloco(DRIVER:=1,CWORD:=6);
	COMMAND_LIFTER_ENABLE:
		fbenadisloco(DRIVER:=1,CWORD:=47);
	COMMAND_ROTATOR_DISABLE:
		fbenadisloco(DRIVER:=2,CWORD:=6);
	COMMAND_ROTATOR_ENABLE:
		fbenadisloco(DRIVER:=2,CWORD:=47);
	COMMAND_PF_ENADIS:
		robotdata.pfEnableContactor:=NOT robotdata.pfEnableContactor;
	COMMAND_DRIVER_ENADIS:
		robotdata.driverContactor:=NOT robotdata.driverContactor;
	STARTSTOP_CHARGE:
		robotdata.chargerContactor:=NOT robotdata.chargerContactor;
	COMMAND_CANCEL_COMMAND:
		cancelcommand:=true;
	COMMAND_RESET_ERRORS:
		fbreseterrors();
	COMMAND_TOGGLE_CONT:
		robotdata.controller:=ABS(robotdata.controller-1);
		st_command.command:=0;
		robotdata.activeState:=CONT_TOGGLE_ENDED;
	COMMAND_SET_MOTIONLIMITS:
		ACCELERATION_LIMIT:=st_command.acc;
		JERK_LIMIT:=st_command.jerk;
		SPEED_LIMIT:=st_command.spd;
	END_CASE
	
CASE st_command.command OF
	3:
    	forwardCommand:=st_command.distance;
    	userCommand:=4;
	10:
    	IF(st_command.direction=0) THEN userCommand:=1;
    	ELSIF(st_command.direction=1)then userCommand:=2;
		END_IF
		
END_CASE
ELSIF topic='STOPPER' then
	robotdata.motorCword[0]:=43;
	robotdata.motorCword[1]:=43;
END_IF
OnMqttMessage := S_OK;
END_METHOD

END_FUNCTION_BLOCK

// ---- POUs/reset_errors.TcPOU
FUNCTION_BLOCK PUBLIC reset_errors
VAR
	 bStart          : BOOL := TRUE;
	 fbTimer         : TON;
	 fbTrigger       : R_TRIG;
	 tTimerValue     : TIME := T#1S;
END_VAR

GVL.robotdata.motorCword[0]:=128;
GVL.robotdata.motorCword[1]:=128;
GVL.robotdata.motorCword[2]:=128;
GVL.robotdata.motorCword[3]:=128;
fbTimer(IN := bStart, PT := tTimerValue);
motion_index:=max_location;
robotdata.motion_status:=MOTION_ENDED;
robotdata.Position_Velocity.Locomotion_1_target_velocity:=0;
robotdata.Position_Velocity.Locomotion_2_target_velocity:=0;
robotdata.Position_Velocity.Rotator_target_velocity:=0;
robotdata.Position_Velocity.Lifter_target_position:=robotdata.Position_Velocity.Lifter_position_actual_value;
robotdata.Position_Velocity.Rotator_target_position:=robotdata.Position_Velocity.Rotator_position_actual_value;

st_command.command:=0;
robotdata.activecommand:=0;

END_FUNCTION_BLOCK

// ---- POUs/enable_disable_driver.TcPOU
FUNCTION_BLOCK PUBLIC enable_disable_driver
VAR_INPUT
	DRIVER:INT;
	CWORD:INT;
END_VAR

IF(DRIVER=0) THEN
	GVL.robotdata.motorCword[0]:=CWORD;
	GVL.robotdata.motorCword[1]:=CWORD;
ELSIF DRIVER=1 THEN
	GVL.robotdata.motorCword[2]:=CWORD;
ELSIF DRIVER=2 THEN
	GVL.robotdata.motorCword[3]:=CWORD;
END_IF

st_command.command:=0;
robotdata.activecommand:=0;

END_FUNCTION_BLOCK

// ---- POUs/kalman/robotAutomation.TcPOU
PROGRAM robotAutomation
VAR
END_VAR

    IF(missionCompleted=1)THEN          // Same as StopMovement??}
      CASE userCommand OF
		  1,2,3:
		  	robotdata.activeState:=TURN_ENDED;
		4,5:
		robotdata.activeState:=MOVE_ENDED;
	  END_CASE
      robot_state:=0;
      modeEnable:=0;
      userCommand:=0;
    
    ELSIF(robot_state=0)THEN
      CASE userCommand OF
        1:  
          robot_state:=1;
          AngPosCommand:=myfmod(idealAngle+90,360)-180;
          modeEnable:=1;
          robotdata.motion_status:=MOTION_ANGLE;
          xGoal:=PosFdbckX;
          yGoal:=PosFdbckY;      
         2:          //TURN LEFT
          robot_state:=2;
          AngPosCommand:=myfmod(idealAngle-90,360)-180;
          modeEnable:=2;
          robotdata.motion_status:=MOTION_ANGLE;
          xGoal:=PosFdbckX;
          yGoal:=PosFdbckY;
         3:          //TURN BACK
          robot_state:=3;
          AngPosCommand:=myfmod(idealAngle+180,360);
          IF (AngPosCommand = 270) THEN
			AngPosCommand := -90;
			END_IF
          modeEnable:=3;
          robotdata.motion_status:=MOTION_ANGLE;
          xGoal:=PosFdbckX;
          yGoal:=PosFdbckY;
            
        4:           //FORWARD   
          robot_state:=4;
          robotdata.motion_status:=MOTION_ONGOING;
          xStart:=LREAL_TO_INT(PosFdbckX);
          yStart:=LREAL_TO_INT(PosFdbckY);
          xGoal:=xStart+COS(idealAngle*PI/180) * forwardCommand;
          yGoal:=yStart+SIN(idealAngle*PI/180) * forwardCommand;
          IF (xGoal >= 7) THEN
			xGoal := 7;
			END_IF
          IF (xGoal <= 0) THEN
			xGoal := 0;
		END_IF
          IF (yGoal >= 8) THEN 
			yGoal := 8;
			END_IF
          IF (yGoal <= 0) THEN 
			yGoal := 0;
			END_IF

          modeEnable:=4;
          
        5: // BACKWARD
          robot_state:=5;
          robotdata.motion_status:=MOTION_ONGOING;
          xStart:=LREAL_TO_INT(PosFdbckX);
          yStart:=LREAL_TO_INT(PosFdbckY);
          xGoal:=xStart - COS(idealAngle*PI/180) * forwardCommand;
          yGoal:=yStart - SIN(idealAngle*PI/180) * forwardCommand;
          IF (xGoal >= 7) THEN xGoal := 7; END_IF
          IF (xGoal <= 0) THEN xGoal := 0; END_IF
          IF (yGoal >= 8) THEN yGoal := 8; END_IF
          IF (yGoal <= 0) THEN yGoal := 0; END_IF
			  
		

          modeEnable:=5;
          
      END_CASE
    END_IF

END_PROGRAM

// ---- POUs/kalman/myfmod.TcPOU
FUNCTION myfmod : LREAL
VAR_INPUT
	x,y:LREAL;
END_VAR
VAR
END_VAR

myfmod:=x-floor(x/y)*y;

END_FUNCTION

// ---- POUs/MAIN.TcPOU
PROGRAM MAIN


VAR
	FB_SET_ENCODER_ODEOMETRY:set_encoder_odeometry();
	FB_DRIVE_MOTORS:DriveMotors();
	gyroZSum:LREAL:=0;
	accXSum:LREAL:=0;
	FB_CONTROLLER:motion_controller;
	dontcontinue:BOOL:=FALSE;
	currtime:ULINT;
	datediff:ULINT;
	fb_kalmaninit:kalmanInit;
	fb_kalmanStep:kalmanStep;
	fb_kalmanController:kalmanController;

END_VAR

//LATE/ERROR KONTROLÜ
IF(calibrationCount<500) THEN
      gyroZSum:=gyroZSum+robotdata.imu_state.hr_gyro_z;
      accXSum:=accXSum+robotdata.imu_state.hr_acc_x;
      calibrationCount:=calibrationCount+1;
ELSIF (calibrationCount=500)THEN
      gyroZmean:=gyroZSum/500;
      accXmean:=accXSum/500;
      calibrationCount:=calibrationCount+1;
    END_IF
	
IF NOT KALMAN_INITIALIZED AND pf_valid=1 THEN
	fb_kalmaninit();
	KALMAN_INITIALIZED:=TRUE;
END_IF
robotdata.batteryVoltage:=DINT_TO_REAL(batteryVoltageINT)/1000;
currtime:=F_GetSystemTime() ;
datediff:=(currtime/10000)-ads_lasttime;
IF (currtime-lastqrtime > NO_QR_TIMEOUT OR (pf_valid=1 AND robotdata.qr_x=0 AND  robotdata.qr_angle=0 AND raw_qr_tag=0 AND robotdata.qr_y=0)) AND robotdata.motion_status=MOTION_ENDED THEN
	robotdata.motion_status:=QRCAM_ERROR;
	pf_valid:=0;
	robotdata.activestate:=QRCAM_ERROR;
ELSIF currtime-lastqrtime < NO_QR_TIMEOUT  AND robotdata.motion_status=QRCAM_ERROR THEN
	robotdata.motion_status:=MOTION_ENDED;
	robotdata.activestate:=MOTION_ENDED;
END_IF

IF currtime-lastqrtagtime > NO_QR_TIMEOUT AND robotdata.motion_status=MOTION_ENDED THEN
	robotdata.activestate:=LOST;
ELSIF currtime-lastqrtagtime < NO_QR_TIMEOUT AND robotdata.activestate=LOST THEN
	robotdata.activestate:=MOTION_ENDED;
END_IF
IF (currtime/10000)-ads_lasttime > NO_ADS_TIMEOUT AND (robotdata.motion_status>PLC_ERROR OR robotdata.motion_status=MOTION_ENDED) THEN
	robotdata.motion_status:=PLC_ERROR;
	robotdata.activestate:=PLC_ERROR;
ELSIF (currtime/10000)-ads_lasttime < NO_ADS_TIMEOUT AND (robotdata.motion_status=PLC_ERROR) THEN
robotdata.motion_status:=MOTION_ENDED;
robotdata.activestate:=MOTION_ENDED;
END_IF
IF(robotdata.motorError[0]+robotdata.motorError[1]+robotdata.motorError[2]+robotdata.motorError[3]>0) AND robotdata.motion_status=MOTION_ENDED  THEN
	robotdata.motion_status:=MOTOR_ERROR;
ELSIF(robotdata.motorError[0]+robotdata.motorError[1]+robotdata.motorError[2]+robotdata.motorError[3]=0 AND robotdata.motion_status=MOTOR_ERROR)THEN
robotdata.motion_status:=MOTION_ENDED;
END_IF
FB_SET_ENCODER_ODEOMETRY();
IF(KALMAN_INITIALIZED)THEN
	fb_kalmanStep();
END_IF

robotdata.encoderx_rel:=robotdata.encoder_x-LREAL_TO_DINT(robotdata.encoder_x);
robotdata.encodery_rel:=robotdata.encoder_y-LREAL_TO_DINT(robotdata.encoder_y);
PosFdbckX_Rel:=PosFdbckX-LREAL_TO_DINT(PosFdbckX);
PosFdbckY_Rel:=PosFdbckY-LREAL_TO_DINT(PosFdbckY);
robotdata.imux_rel:=robotdata.imu_state.imu_x-LREAL_TO_DINT(robotdata.imu_state.imu_x);
robotdata.imuy_rel:=robotdata.imu_state.imu_y-LREAL_TO_DINT(robotdata.imu_state.imu_y);

IF(CONTROLLER_TYPE=0)THEN
	IF(pf_valid=0)THEN
		robotdata.robot_x:=robotdata.encoder_x;
		robotdata.robot_y:=robotdata.encoder_y;
		robotdata.robot_yaw:=robotdata.imu_state.imu_euler;
		winnerEvaluated:=FALSE;
	END_IF
	FB_CONTROLLER();
	FB_DRIVE_MOTORS();
ELSIF(CONTROLLER_TYPE=1 AND KALMAN_INITIALIZED) THEN
	robotdata.robot_x:=PosFdbckX;
	robotdata.robot_y:=PosFdbckY;
	robotdata.robot_yaw:=robotAngle *PI/180;
	fb_kalmanController();
END_IF

END_PROGRAM

// ---- POUs/set_encoder_odeometry.TcPOU
FUNCTION_BLOCK PUBLIC set_encoder_odeometry
VAR
	
	current_x_state:LREAL;
	current_y_state:LREAL;
	radius:LREAL;
	icc_x:LREAL;
	icc_y:LREAL;
	yaw_prev:LREAL;
	
END_VAR

	slave0_speed := robotdata.Position_Velocity.Locomotion_1_actual_velocity;       
	slave1_speed := robotdata.Position_Velocity.Locomotion_2_actual_velocity;       
	slave1_speed:=-1 * slave1_speed;
	robotdata.encoder_omega := (slave1_speed - slave0_speed) * RPM2MSN / ((ROBOT_RADIUS) * 2.0); //angular velocity
	robotdata.encoder_v:= (slave1_speed + slave0_speed) * RPM2MSN / 2.0; // linear velocity


	robotdata.encoder_slave0_speed := slave0_speed * RPM2MSN;
	robotdata.encoder_slave1_speed := slave1_speed * RPM2MSN;
	IF (slave0_speed<>slave1_speed) THEN
	
		current_x_state := robotdata.encoder_x;
		current_y_state := robotdata.encoder_y;

		radius:= (ROBOT_RADIUS) * (slave1_speed + slave0_speed) / (slave1_speed - slave0_speed);
		icc_x := robotdata.encoder_x - (radius * SIN(robotdata.encoder_yaw)); //ICC
		icc_y := robotdata.encoder_y + (radius * COS(robotdata.encoder_yaw)); //ICC
		 IF(pf_valid=0)THEN
			robotdata.encoder_x := ((current_x_state - icc_x) * COS(robotdata.encoder_omega * GVL.PLC_CYCLE)) - (current_y_state - icc_y) * SIN(robotdata.encoder_omega * PLC_CYCLE) + icc_x;
			robotdata.encoder_y := ((current_x_state - icc_x) * SIN(robotdata.encoder_omega * GVL.PLC_CYCLE)) + (current_y_state - icc_y) * COS(robotdata.encoder_omega * PLC_CYCLE) + icc_y;
		END_IF
		IF(pf_valid=1)THEN
			robotdata.encoder_yaw := robotdata.qr_yaw;
		ELSE
		robotdata.encoder_yaw := robotdata.encoder_yaw + (robotdata.encoder_omega * PLC_CYCLE); //heading
		END_IF
	

	
	ELSE
	
		robotdata.encoder_x := robotdata.encoder_x+(robotdata.encoder_v * PLC_CYCLE * COS(robotdata.encoder_yaw)); // x coordinate
		robotdata.encoder_y := robotdata.encoder_y+(robotdata.encoder_v * PLC_CYCLE * SIN(robotdata.encoder_yaw)); // y coordinate
	END_IF

END_FUNCTION_BLOCK

// ---- POUs/DriveMotors.TcPOU
FUNCTION_BLOCK PUBLIC DriveMotors
VAR
END_VAR

IF (robotdata.motion_status = MOTION_ANGLE) THEN
		robotdata.Position_Velocity.Locomotion_1_target_velocity := motion_left[motion_index];
		robotdata.Position_Velocity.Locomotion_2_target_velocity:= motion_right[motion_index];
		IF(robotdata.lifterDistance>LIFTER_UP) THEN
			//robotdata.Position_Velocity.Rotator_Target_Position:= motion_rotator[motion_index];
			robotdata.Position_Velocity.Rotator_Target_Velocity:=LREAL_TO_DINT(-3.16*motion_right[motion_index]);
		END_IF
		motion_index:=motion_index+1;
		IF (motion_index = max_location) THEN
			robotdata.motion_status := MOTION_ENDED;
			robotdata.activeState:=TURN_ENDED;
			robotdata.Position_Velocity.Locomotion_1_target_velocity:= 0;
			robotdata.Position_Velocity.Locomotion_2_target_velocity:= 0;
			robotdata.Position_Velocity.Rotator_Target_Velocity:=0;
		END_IF
ELSIF (robotdata.motion_status = MOTION_ONGOING) THEN
	
		robotdata.Position_Velocity.Locomotion_1_target_velocity := motion_left[motion_index];
		robotdata.Position_Velocity.Locomotion_2_target_velocity:= -1*motion_right[motion_index];
		motion_index:=motion_index+1;
		IF (motion_index = max_location) THEN
			robotdata.motion_status := MOTION_ENDED;
				robotdata.activeState:=MOVE_ENDED;
			robotdata.Position_Velocity.Locomotion_1_target_velocity:= 0;
			robotdata.Position_Velocity.Locomotion_2_target_velocity:= 0;
		END_IF

ELSIF (robotdata.motion_status = MOTION_LIFTER) THEN
	IF(motion_index = max_location ) OR (robotdata.activeState=LIFT_UP AND robotdata.lifterDistance>LIFTER_UP_LIMIT) OR(robotdata.activeState=LIFT_DOWN AND robotdata.lifterDistance<LIFTER_DOWN_LIMIT)  THEN
		IF(robotdata.activeState=LIFT_UP) THEN
		 robotdata.lifter:=60;
		ELSE
			robotdata.lifter:=0;
		END_IF
		robotdata.motion_status:=MOTION_ENDED;
		robotdata.activeState:=LIFT_ENDED;
		motion_index:=max_location;
	ELSE
		robotdata.Position_Velocity.Lifter_target_position := motion_lift[motion_index];
		motion_index:=motion_index+1;
	END_IF
ELSIF (robotdata.motion_status = MOTION_ROTATE) THEN
	IF(motion_index = max_location )THEN
		robotdata.motion_status:=MOTION_ENDED;
		robotdata.activeState:=ROTATE_ENDED;
		motion_index:=max_location;
		robotdata.Position_Velocity.Rotator_Target_Velocity:=0;
		ELSE
		//robotdata.Position_Velocity.Rotator_Target_Position:= motion_rotator[motion_index];
		robotdata.Position_Velocity.Rotator_Target_Velocity:= motion_rotator[motion_index];
		motion_index:=motion_index+1;
	END_IF		
END_IF

END_FUNCTION_BLOCK

// ---- POUs/motion_controller.TcPOU
FUNCTION_BLOCK PUBLIC motion_controller
VAR
  vc:LREAL;
  wc:LREAL;

  vreff:LREAL;
  qrError:LREAL ;
  imu_local_y:LREAL ;
  enc_local_y:LREAL ;
  local_x:LREAL:=0;
  local_y:LREAL:=0;
  
  stabilization_lateral:LREAL;
  motion_direction_sign:INT:=-1;
  reference_position:LREAL := 0.0;
  reference_velocity:LREAL := 0.0;
  ref_temp:LREAL := 0.0;
  cos_angle_diff:LREAL;
  k_xx:LREAL;
  k_xi:LREAL;
  err_int:LREAL;
  err_x:LREAL;
  errY:LREAL;
  
  errTheta:LREAL;
 

 wccoeff:INT;
 l_wh_lin_speed:LREAL;
 r_wh_lin_speed:LREAL;
 rr:LREAL:=0;
 omega:LREAL:=0;
 left_arc:LREAL:=0;
 right_arc:LREAL:=0;
 l_arc_dec:DINT:=0;
 r_arc_dec:DINT:=0;
 omegasign:INT;
 vsign:INT;
 rpmL:DINT;
 rpmR:DINT;
END_VAR

 
  IF(robotdata.robot_direction MOD 2 =0) THEN
    local_x := robotdata.encoder_x;
    local_y := robotdata.robot_y;
    IF(imuYwins=0) THEN
      local_y := robotdata.encoder_y;
	END_IF
    imu_local_y:=robotdata.imu_state.imu_y;
    enc_local_y:=robotdata.encoder_y;
    IF(imuYwins=1) THEN
      local_y := robotdata.imu_state.imu_y;
	END_IF
    //local_y:=PosFdbckY;
    IF(robotdata.qr_tag>0) THEN
      qrError:=(-1)*(robotdata.qr_y)/1000;
	END_IF
  ELSIF(robotdata.robot_direction MOD 2 = 1) THEN
  
    local_x := robotdata.encoder_y;
    local_y := robotdata.robot_x;
    IF(imuXwins=0)THEN
      local_y := robotdata.encoder_x;
	END_IF
  
    imu_local_y:=robotdata.imu_state.imu_x;
    enc_local_y:=robotdata.encoder_y;
 
    IF(imuXwins=1)THEN
      local_y := robotdata.imu_state.imu_x;
	END_IF
	//local_y:=PosFdbckX;
    IF(robotdata.qr_tag>0)THEN
      qrError:=(-1)*(robotdata.qr_x)/1000;
	END_IF
  END_IF

  stabilization_lateral := GRID_DIM *LREAL_TO_DINT(local_y/GRID_DIM);
 
  IF(robotdata.robot_direction = 0  OR robotdata.robot_direction = 3) THEN
    motion_direction_sign := 1;
  END_IF
  IF(robotdata.robot_direction = 0 OR robotdata.robot_direction = 1)THEN
    lateral_direction_sign := 1;
  ELSE
	  lateral_direction_sign := -1;
  END_IF
  
  
  // ERROR MODEL IMPLEMENTATION
  
    reference_position :=  ABS(motion_direction_sign * (motion[motion_index] * DEC2M) + local_x_before_motion);//local_x_before_motion move da set ediliyor 
    ref_temp := reference_position;
    reference_velocity :=  ABS(motion_vel[motion_index]);
  
  //this is temporary, will be optimized
  cos_angle_diff := 0;
  IF(robotdata.robot_direction = 1)THEN
    cos_angle_diff := PI/2.0;
  ELSIF (robotdata.robot_direction = 3)THEN
    cos_angle_diff := -PI/2.0;
  END_IF

  vreff := reference_velocity;

  //vc = vreff / cos(feedback_state->yaw_state+cos_angle_diff) + (copysign(1.0, err_x) * MIN(ACCELERATION_LIMIT * (g_app_config->ts_rollout), fabs(err_x)));
  vc := vreff;
  vc := MIN(ABS(vc), SPEED_LIMIT * 1.10);

  // Stanley - Y controller
  errY :=  lateral_direction_sign*(stabilization_lateral - local_y);
  imu_local_y:=lateral_direction_sign*(stabilization_lateral - imu_local_y);
  enc_local_y:=lateral_direction_sign*(stabilization_lateral - enc_local_y);
  //double current_yaw_deg =feedback_state->yaw_state * 180.0 / M_PI;
  
	IF(FALSE and imuAngwins)THEN
  		current_yaw_deg :=LMOD(robotdata.imu_state.imu_euler+2 * PI,2*PI)*180/PI;
	ELSE
		current_yaw_deg :=LMOD(robotdata.encoder_yaw+2 * PI,2*PI)*180/PI;
	END_IF
   
  IF(robotdata.qr_tag>0)THEN
    current_yaw_deg:= LMOD(robotdata.qr_yaw+2 * PI,2*PI)*180/PI;
  END_IF
  stabilization_yaw_deg:=detectStabilizedAngle(current_yaw:=current_yaw_deg);
 // printf("%d,%lf,%lf,%lf\n",robot_direction,stabilization_yaw_deg,current_yaw_deg,feedback_state->local_yaw_error);
  errTheta := stabilization_yaw_deg - current_yaw_deg;
  IF(ABS(errTheta)>30 AND robotdata.motion_status=MOTION_ONGOING)THEN
    errTheta:=0;
  END_IF
  
  IF(robotdata.qr_tag>0 AND ABS(qrError)>0) THEN
    errY:=lateral_direction_sign*qrError;
  END_IF
   robotdata.deviation_y:=errY;
  robotdata.deviation_yaw:=errTheta*PI/180;
  //printf("%lf,%lf,%lf\n",stabilization_yaw_deg,current_yaw_deg,feedback_state->local_yaw_error);
 
  
  
  robotdata.wc1 := (KpY*errY) * OMEGA_DIFF_MAX;
   
  // printf("Stab/Err:%lf/%lf ",stabilization_yaw_deg,imueuler);
   away:=-1 * TOWARDS_COEFF;
   IF(
   (robotdata.robot_direction=0  AND errY<0 AND current_yaw_deg >0 AND current_yaw_deg<90)OR
   (robotdata.robot_direction=0  AND errY>0 AND current_yaw_deg >270 AND current_yaw_deg<359.9)OR
   (robotdata.robot_direction=1  AND errY<0 AND current_yaw_deg >270 AND current_yaw_deg<359.9)OR
   (robotdata.robot_direction=1  AND errY>0 AND current_yaw_deg <270 AND current_yaw_deg>180)OR
   (robotdata.robot_direction=2  AND errY<0 AND current_yaw_deg >180 AND current_yaw_deg<270)OR
   (robotdata.robot_direction=2  AND errY>0 AND current_yaw_deg >90 AND current_yaw_deg<180)OR
   (robotdata.robot_direction=3  AND errY<0 AND current_yaw_deg >90 AND current_yaw_deg<180)OR
   (robotdata.robot_direction=3  AND errY>0 AND current_yaw_deg >0 AND current_yaw_deg<90))THEN
   away:=AWAY_COEFF;
   END_IF
   IF(robotdata.wc1<0) THEN 
	wccoeff:=-1;
   ELSE
	wccoeff:=1;
   END_IF
  
   robotdata.wc2:=(wccoeff*away*KpTht*ABS(errTheta));
   //if(copysign(1,wc)!=copysign(1,wc2))
   // wc=0;
  //else
   wc:=robotdata.wc1+robotdata.wc2;   

  IF ( (pf_valid=1 AND ABS(errY)<Y_DEV_THRESHOLD) OR (pf_valid=0 AND ABS(errY)<Y_DEV_THRESHOLD/2) OR ABS(vc)<0.2) AND away<0 THEN
    wc:=0;
  END_IF  
    
  //wc=wc*fabs(feedback_state->v_state/SPEED_LIMIT); 
  

 

  
  controller_coeff:=wc;


  l_wh_lin_speed := ((2*vc) - (wc * 2.0 * (ROBOT_RADIUS))) / (2.0);
  r_wh_lin_speed := ((2*vc) + (wc * 2.0 * (ROBOT_RADIUS))) / (2.0);
  IF(l_wh_lin_speed>2*SPEED_LIMIT) THEN l_wh_lin_speed:=1.5*SPEED_LIMIT;END_IF;
  IF(r_wh_lin_speed>2*SPEED_LIMIT)THEN r_wh_lin_speed:=1.5*SPEED_LIMIT;END_IF;
  


 

  IF (l_wh_lin_speed <> r_wh_lin_speed) THEN
  
    rr := ABS((robot_radius) * ((r_wh_lin_speed + l_wh_lin_speed) / (r_wh_lin_speed - l_wh_lin_speed)));
    omega := (r_wh_lin_speed - l_wh_lin_speed) / ((robot_radius) * 2.0);
	IF(omega<0) THEN 
	omegasign:=-1;
	ELSE
		omegasign:=1;
	END_IF
    left_arc := (rr - (omegasign * (robot_radius))) * (ABS(omega) * (PLC_CYCLE));
    right_arc := (rr + (omegasign * (robot_radius))) * (ABS(omega) * (PLC_CYCLE));

    //printf("vl |> %lf \t vr |> %lf\n", l_wh_lin_speed, r_wh_lin_speed);

    l_arc_dec := LREAL_TO_DINT(left_arc * M2DEC);
    r_arc_dec := LREAL_TO_DINT(right_arc * M2DEC);
  
  else
     l_arc_dec := LREAL_TO_DINT(l_wh_lin_speed * (PLC_CYCLE) * M2DEC);
    r_arc_dec :=  LREAL_TO_DINT(r_wh_lin_speed * (PLC_CYCLE) * M2DEC);
  END_IF

  
  IF (robotdata.controller=1 AND robotdata.motion_status = MOTION_ONGOING AND wc<>0) THEN
  	IF(reference_velocity<0) THEN 
	vsign:=-1;
	ELSE
	vsign:=1;	
	END_IF
    rpmL:= LREAL_TO_DINT(vsign * LREAL_TO_DINT((REDUCER_RATIO*l_wh_lin_speed*60)/(2*PI*WHEEL_RADIUS)));
    rpmR:= LREAL_TO_DINT(vsign * LREAL_TO_DINT((REDUCER_RATIO*r_wh_lin_speed*60)/(2*PI*WHEEL_RADIUS)));
   
    motion_left[motion_index] :=rpmL;
    motion_right[motion_index]:=rpmR;
  END_IF

END_FUNCTION_BLOCK

// ---- POUs/detectStabilizedAngle.TcPOU
FUNCTION detectStabilizedAngle:LREAL
VAR_INPUT
	current_yaw:LREAL;
END_VAR
VAR_OUTPUT
	stab_angle:LREAL;
END_VAR
VAR
END_VAR

IF ((current_yaw >= 0 AND current_yaw <= 45))THEN
      stab_angle := 0;
 	robotdata.robot_direction := 0;
    
	ELSIF ((current_yaw >= 315 AND current_yaw <= 360))THEN
      stab_angle := 360;
	robotdata.robot_direction := 0;
    
    ELSIF ( (current_yaw >= 270 AND current_yaw <= 315)OR (current_yaw >= 225 AND current_yaw <= 270))  THEN
      stab_angle := 270;
     robotdata.robot_direction := 1;
    ELSIF ((current_yaw <= 225 AND current_yaw >= 180)OR(current_yaw >= 135 AND current_yaw <= 180))  THEN
      stab_angle := 180;
     robotdata.robot_direction := 2;
    
    ELSE 
     stab_angle := 90;
	  robotdata.robot_direction := 3;
    END_IF
	detectStabilizedAngle:=stab_angle;

END_FUNCTION

// ---- POUs/kalman/kalmanInit.TcPOU
FUNCTION_BLOCK kalmanInit
VAR_INPUT
END_VAR
VAR_OUTPUT
END_VAR
VAR
	tmp0:ARRAY[0..2,0..2] OF LREAL;
	Ft:ARRAY[0..2,0..2] OF LREAL;
	tmp:ARRAY[0..2,0..0] OF LREAL;
	tmp1:ARRAY[0..2,0..2] OF LREAL;

	
END_VAR

  mulmat(F_kalman1,x_kalman1,tmp,3,3,1);
  mulmat(I,tmp,x_kalman1,3,3,1);
  x_kalman2[0,0]:=-1 * robotdata.qr_angle * 0.1;
  mulmat(F_kalman1, P_kalman1 ,tmp0, 3, 3, 3);
  transpose(F_kalman1,Ft, 3, 3);
  mulmat(tmp0, Ft, P_kalman1, 3, 3, 3);
  accum(P_kalman1, Q_kalman1, 3, 3);

  mulmat(F_kalman2,x_kalman2,tmp,3,3,1);
  mulmat(I,tmp,x_kalman2,3,3,1);

  mulmat(F_kalman2, P_kalman2 ,tmp0, 3, 3, 3);
  transpose(F_kalman2,Ft, 3, 3);
  mulmat(tmp0, Ft, P_kalman2, 3, 3, 3);
  accum(P_kalman2, Q_kalman2, 3, 3);

  F_kalman3[0,2]:= -1*x_kalman1[0,0]*COS(x_kalman2[0,0]*PI/180)*PLC_CYCLE;
  F_kalman3[1,2]:= -1*x_kalman1[0,0]*SIN(x_kalman2[0,0]*PI/180)*PLC_CYCLE;
  
  x_kalman3[0,0]:=qr_xstate+x_kalman1[0,0]*COS(x_kalman2[0,0]*PI/180)*PLC_CYCLE;
  x_kalman3[1,0]:=qr_ystate+x_kalman1[0,0]*SIN(x_kalman2[0,0]*PI/180)*PLC_CYCLE;
  x_kalman3[2,0]:=(-1 * robotdata.qr_angle * 0.1)+x_kalman2[1,0]*PLC_CYCLE;

  //P_kalman3 = Fk_kalman3*P_kalman3*Fk_kalman3'+Q_kalman3;
  transpose(F_kalman3,Ft,3,3);
  mulmat(F_kalman3,P_kalman3,tmp0,3,3,3);//tmp0=k_kalman3*P_kalman3
  mulmat(tmp0,Ft,P_kalman3,3,3,3);//P_kalman3=tmp0*Fk_kalman3
  accum(P_kalman3,Q_kalman3,3,3);//P_kalman3=tmp0*Fk_kalman3+Q_kalman3
  
  kalman12_x :=qr_xstate;
  kalman12_y := qr_ystate;

END_FUNCTION_BLOCK

// ---- POUs/kalman/mulmat.TcPOU
FUNCTION mulmat : BOOL
VAR_IN_OUT
	a:ARRAY[*,*] OF LREAL;
	b:ARRAY[*,*] OF LREAL;
	c:ARRAY[*,*] OF LREAL;
END_VAR
VAR_INPUT
	arows,acols,bcols:SINT;
END_VAR
VAR
	i, j,l:SINT;
END_VAR

FOR i:=0 TO arows-1 DO
        FOR j:=0 TO bcols-1 DO 
            c[i,j] := 0;
            FOR l:=0 TO acols-1 DO
                c[i,j] := c[i,j]+a[i,l] * b[l,j];
			END_FOR
		END_FOR
END_FOR
mulmat:=TRUE;

END_FUNCTION

// ---- POUs/kalman/transpose.TcPOU
FUNCTION transpose : BOOL
VAR_IN_OUT
	a,att:ARRAY[*,*] OF LREAL;
END_VAR
VAR_INPUT
	m,n:SINT;
END_VAR
VAR
	i,j:SINT;
END_VAR


    FOR i:=0 TO m-1 DO 
        FOR j:=0 TO n-1 DO 
            att[j,i] := a[i,j];
        END_FOR
	END_FOR
	transpose:=true;

END_FUNCTION

// ---- POUs/kalman/accum.TcPOU
FUNCTION accum : BOOL
VAR_IN_OUT
	a,b:ARRAY[*,*] OF LREAL;
END_VAR
VAR_INPUT
	m,n:SINT;
END_VAR
VAR
	i,j:SINT;
END_VAR

		
FOR i:=0 TO m-1 DO
        FOR j:=0  TO n-1 DO 
            a[i,j] := a[i,j]+b[i,j];
			END_FOR
	END_FOR
	accum:=true;

END_FUNCTION

// ---- POUs/kalman/kalmanStep.TcPOU
FUNCTION_BLOCK kalmanStep
VAR_INPUT
END_VAR
VAR_OUTPUT
END_VAR
VAR
tmp0:ARRAY[0..2,0..2] OF LREAL;
tmp00:ARRAY[0..2,0..2] OF LREAL;
tmp00s:ARRAY[0..2,0..2] OF LREAL;
tmp00t:ARRAY[0..2,0..2] OF LREAL;
tmp000:ARRAY[0..2,0..2] OF LREAL;
Ft:ARRAY[0..2,0..2] OF LREAL;
Ht:ARRAY[0..2,0..1] OF LREAL;
Ht3:ARRAY[0..2,0..2] OF LREAL;
tmp1:ARRAY[0..2,0..1] OF LREAL;
tmp2:ARRAY[0..1,0..2] OF LREAL;
tmp3:ARRAY[0..1,0..1] OF LREAL;
tmp4:ARRAY[0..1,0..1] OF LREAL;
tmp5:ARRAY[0..1] OF LREAL;
tmp6:ARRAY[0..1,0..0] OF LREAL;
tmp7:ARRAY[0..1,0..0] OF LREAL;
tmp8:ARRAY[0..2,0..0] OF LREAL;
tmp5_3:ARRAY[0..2] OF LREAL;
tmp1_3,tmp2_3,tmp3_3,tmp4_3,Kt3:ARRAY[0..2,0..2] OF LREAL;
tmp6_3,tmp7_3:ARRAY[0..2] OF LREAL;
Kt:ARRAY[0..1,0..2] OF LREAL;
	 fb_localization:localization;
END_VAR

  fb_localization();
  linSpdFdbckRobot := (rightWheelFdbck+leftWheelFdbck)*2*PI/60*wheel_radius/2;
  posTheta_wrt_robot_enc :=((-1*Locomotion_2_actual_pos - Locomotion_1_actual_pos)/10000)*360*wheel_radius/(2*robot_radius)/reducer_ratio + (-1*robotdata.qr_angle * 0.1); 
  //posTheta_wrt_robot_enc :=robotdata.encoder_omega*180/PI;
  //linSpdFdbckRobot :=robotdata.encoder_v; 
  z_kalman1[0,0]:=linSpdFdbckRobot;
  z_kalman1[1,0]:=robotdata.imu_state.hr_acc_x;
  z_kalman2[0,0]:=posTheta_wrt_robot_enc;
  z_kalman2[1,0]:=(robotdata.imu_state.hr_gyro_z)*180/PI;

  kalman12_x := kalman12_x + x_kalman1[0,0]*COS(x_kalman2[0,0]*PI/180)*PLC_CYCLE;
  kalman12_y := kalman12_y + x_kalman1[0,0]*SIN(x_kalman2[0,0]*PI/180)*PLC_CYCLE;
  z_kalman3[0,0] :=qr_xstate;
  z_kalman3[1,0] := qr_ystate;
  z_kalman3[2,0] := -1*robotdata.qr_angle * 0.1;
      
  IF (pf_valid=0)THEN
        H_kalman3[0,0]:=0;H_kalman3[0,1]:=0;H_kalman3[0,2]:=0;
        H_kalman3[1,0]:=0;H_kalman3[1,1]:=0;H_kalman3[1,2]:=0;
        H_kalman3[2,0]:=0;H_kalman3[2,1]:=0;H_kalman3[2,2]:=0;
  
    else
        H_kalman3[0,0]:=1;H_kalman3[0,1]:=0;H_kalman3[0,2]:=0;
        H_kalman3[1,0]:=0;H_kalman3[1,1]:=1;H_kalman3[1,2]:=0;
        H_kalman3[2,0]:=0;H_kalman3[2,1]:=0;H_kalman3[2,2]:=1;
      END_IF
      

//************************KALMAN - 1****************************************************************/

    transpose(H_kalman1, Ht, 2, 3);
    mulmat(P_kalman1, Ht, tmp1, 3, 3, 2);

    mulmat(H_kalman1, P_kalman1, tmp2, 2, 3, 3);
    mulmat(tmp2, Ht, tmp3, 2, 3, 2);
    accum(tmp3, R_kalman1, 2, 2);
    IF (cholsl(tmp3, tmp4, tmp5, 2)=1) THEN 
	RETURN;
	END_IF
    mulmat(tmp1, tmp4, K_kalman1, 3, 2, 2);

    //x_kalman1 = x_kalman1 + K_kalman1*(z_kalman1-H_kalman1*x_kalman1);*/
    mulmat(H_kalman1,x_kalman1,tmp6,2,3,1);
    ssub(z_kalman1,tmp6,tmp7,2);
    mulmat(K_kalman1,tmp7,tmp8,3,2,1);
    accum(x_kalman1,tmp8,3,1);
  // P_kalman1 = (eye(3)-K_kalman1*H_kalman1)*P_kalman1*(eye(3)-K_kalman1*H_kalman1)'+K_kalman1*R_kalman1*K_kalman1';*/
  transpose(K_kalman1,Kt,3,2);
  mulmat(R_kalman1,Kt,tmp2,2,2,3);
  mulmat(K_kalman1,tmp2,tmp0,3,2,3);//tmp0=K_kalman1*R_kalman1*K_kalman1'*/
  
  mulmat(K_kalman1,H_kalman1,tmp00,3,2,3);
  sub_mat(I,tmp00,tmp00,3,3);
  transpose(tmp00,tmp00t,3,3);
  mulmat(P_kalman1,tmp00t,tmp00,3,3,3);//tmp00=P_kalman1*(eye(3)-K_kalman1*H_kalman1)'*/
 
  mulmat(K_kalman1,H_kalman1,tmp000,3,2,3);
  sub_Mat(I,tmp000,tmp000,3,3);//tmp000=(eye(3)-K_kalman1*H_kalman1)*/
  
  mulmat(tmp000,tmp00,P_kalman1,3,3,3);//P_kalman1= (eye(3)-K_kalman1*H_kalman1)*P_kalman1*(eye(3)-K_kalman1*H_kalman1)'*/
  accum(P_kalman1,tmp0,3,3);//P_kalman1= (eye(3)-K_kalman1*H_kalman1)*P_kalman1*(eye(3)-K_kalman1*H_kalman1)' + K_kalman1*R_kalman1*K_kalman1'*/
  
//  x_kalman2 = F_kalman2*x_kalman2;*/
  mulmat(F_kalman1,x_kalman1,tmp8,3,3,1);
  mulmat(I,tmp8,x_kalman1,3,3,1);
  //printMat(x_kalman1,3,1);
 // P_kalman2 = F_kalman2*P_kalman2*F_kalman2'+Q_kalman2;*/
  mulmat(F_kalman1, P_kalman1 ,tmp0, 3, 3, 3);
  transpose(F_kalman1,Ft, 3, 3);
  mulmat(tmp0, Ft, P_kalman1, 3, 3, 3);
  accum(P_kalman1, Q_kalman1, 3, 3);

//************************KALMAN - 2****************************************************************/

  //  K_kalman2 = P_kalman2*H_kalman2'*inv(H_kalman2*P_kalman2*H_kalman2'+R_kalman2);   */
  transpose(H_kalman2, Ht, 2, 3);
  mulmat(P_kalman2, Ht, tmp1, 3, 3, 2);
  mulmat(H_kalman2, P_kalman2, tmp2, 2, 3, 3);
  mulmat(tmp2, Ht, tmp3, 2, 3, 2);
  accum(tmp3, R_kalman2, 2, 2);  
    IF (cholsl(tmp3, tmp4, tmp5, 2)=1)THEN
      
      RETURN;
    END_IF
  mulmat(tmp1, tmp4, K_kalman2, 3, 2, 2);
  
  // err_kalman2(1,1) = errorDegreeCalculator(z_kalman2(1), x_kalman2(1)); */
  // err_kalman2(2,1) = z_kalman2 - x_kalman2(2); */
  err_kalman2[0,0] := errorDegreeCalculator(z_kalman2[0,0], x_kalman2[0,0]);
  err_kalman2[1,0] := z_kalman2[1,0] - x_kalman2[1,0];

  // x_kalman2 = x_kalman2 + K_kalman2 * err_kalman2; */
  mulmat(K_kalman2, err_kalman2, tmp8, 3, 2, 1);
  accum(x_kalman2,tmp8,3,1);

  // x_kalman2 = x_kalman2 + K_kalman2*(z_kalman2-H_kalman2*x_kalman2); */ //bu denklem yerine yukarıdaki 3 denklem eklendi
  // mulmat(H_kalman2,x_kalman2,tmp6,2,3,1); 
  // sub(z_kalman2,tmp6,tmp7,2);
  // mulmat(K_kalman2,tmp7,tmp8,3,2,1);
  // accum(x_kalman2,tmp8,3,1);

  // P_kalman2 = (eye(3)-K_kalman2*H_kalman2)*P_kalman2*(eye(3)-K_kalman2*H_kalman2)'+K_kalman2*R_kalman2*K_kalman2';*/
  transpose(K_kalman2,Kt,3,2);
  mulmat(R_kalman2,Kt,tmp2,2,2,3);
  mulmat(K_kalman2,tmp2,tmp0,3,2,3);//tmp0=K_kalman2*R_kalman2*K_kalman2'*/
  
  mulmat(K_kalman2,H_kalman2,tmp00,3,2,3);
  sub_Mat(I,tmp00,tmp00,3,3);
  transpose(tmp00,tmp00t,3,3);
  mulmat(P_kalman2,tmp00t,tmp00,3,3,3);//tmp00=P_kalman2*(eye(3)-K_kalman2*H_kalman2)'*/
 
  mulmat(K_kalman2,H_kalman2,tmp000,3,2,3);
  sub_Mat(I,tmp000,tmp000,3,3);//tmp000=(eye(3)-K_kalman2*H_kalman2)*/
  
  mulmat(tmp000,tmp00,P_kalman2,3,3,3);//P_kalman2= (eye(3)-K_kalman2*H_kalman2)*P_kalman2*(eye(3)-K_kalman2*H_kalman2)'*/
  accum(P_kalman2,tmp0,3,3);//P_kalman2= (eye(3)-K_kalman2*H_kalman2)*P_kalman2*(eye(3)-K_kalman2*H_kalman2)' + K_kalman2*R_kalman2*K_kalman2'*/
  
//**/
  x_kalman2[0,0] := myfmod(x_kalman2[0,0], 360);

//*  x_kalman2 = F_kalman2*x_kalman2;*/
  mulmat(F_kalman2,x_kalman2,tmp8,3,3,1);
  mulmat(I,tmp8,x_kalman2,3,3,1);
  //printMat(x_kalman2,3,1);
 //* P_kalman2 = F_kalman2*P_kalman2*F_kalman2'+Q_kalman2;*/
  mulmat(F_kalman2, P_kalman2 ,tmp0, 3, 3, 3);
  transpose(F_kalman2,Ft, 3, 3);
  mulmat(tmp0, Ft, P_kalman2, 3, 3, 3);
  accum(P_kalman2, Q_kalman2, 3, 3);
  kalLinSpd:= x_kalman1[0,0];
  kalAngSpd:=x_kalman2[1,0];



//*************************KALMAN - 3****************************************************************/

  //  K_kalman3 = P_kalman3*H_kalman3'*inv(H_kalman3*P_kalman3*H_kalman3'+R_kalman3);   */
    transpose(H_kalman3, Ht3, 3, 3);
    mulmat(P_kalman3, Ht3, tmp1_3, 3, 3, 3);
    mulmat(H_kalman3, P_kalman3, tmp2_3, 3, 3, 3);
    mulmat(tmp2_3, Ht3, tmp3_3, 3, 3, 3);
    accum(tmp3_3, R_kalman3, 3, 3);
    IF (cholsl(tmp3_3, tmp4_3, tmp5_3, 3)=1) THEN
      RETURN;
    END_IF 
    
    mulmat(tmp1_3, tmp4_3, K_kalman3, 3, 3, 3);    

    // if(qr_message == 0){
    //   err_kalman3[0] = z_kalman3[0];
    //   err_kalman3[1] = z_kalman3[1];
    //   err_kalman3[2] = errorDegreeCalculator(z_kalman3[2],0);
    // }
    // else{
    //   err_kalman3[0] = z_kalman3[0] -  x_kalman3[0,0];
    //   err_kalman3[1] = z_kalman3[1] -  x_kalman3[0,1];
    //   err_kalman3[2] = errorDegreeCalculator(z_kalman3[2], x_kalman3[0,2]);
    // }

  err_kalman3[0,0] := z_kalman3[0,0] - x_kalman3[0,0];
  err_kalman3[1,0] := z_kalman3[1,0] -	 x_kalman3[1,0];
  err_kalman3[2,0] := errorDegreeCalculator(z_kalman3[2,0], x_kalman3[2,0]); 

  //x_kalman3 = x_kalman3 + K_kalman3*err_kalman3;*/
  mulmat(K_kalman3, err_kalman3, tmp8, 3, 3, 1);
  accum(x_kalman3, tmp8, 3, 1);

  x_kalman3[2,0] := myfmod(x_kalman3[2,0], 360);

  //x_kalman3 = x_kalman3 + K_kalman3*(z_kalman3-H_kalman3*x_kalman3);*/ //bu denklem yerine yukarıdaki 4 denklem eklendi
  //   mulmat(H_kalman3,x_kalman3,tmp6_3,3,3,1);
  //   sub(z_kalman3,tmp6_3,tmp7_3,3);
  //   mulmat(K_kalman3,tmp7_3,tmp8,3,3,1);
  //   accum(x_kalman3,tmp8,3,1);

  // P_kalman3 = (eye(3)-K_kalman3*H_kalman3)*P_kalman3;*/
    mulmat(K_kalman3,H_kalman3,tmp0,3,3,3);
    sub_Mat(I,tmp0,tmp0,3,3);
    mulmat(tmp0,P_kalman3,tmp00,3,3,3);//tmp00=(eye(3)-K_kalman3*H_kalman3)*P_kalman3*/   ////////////////////////
    mulmat(tmp00,I,P_kalman3,3,3,3);

  x_kalman3[0,0] := x_kalman3[0,0] + x_kalman1[0,0]*COS(x_kalman3[2,0]*PI/180)*PLC_CYCLE;
  x_kalman3[1,0] := x_kalman3[1,0] + x_kalman1[0,0]*SIN(x_kalman3[2,0]*PI/180)*PLC_CYCLE;
  IF (pf_valid=0)THEN
  	x_kalman3[2,0] := x_kalman3[2,0] + x_kalman2[1,0]*PLC_CYCLE;
	//x_kalman3[2,0] := LMOD(robotdata.imu_state.imu_euler+2 * PI,2*PI)*180/PI;
  ELSE
	  x_kalman3[2,0] :=-1*robotdata.qr_angle * 0.1;
  END_IF

  IF ( x_kalman3[2,0] >=180 AND x_kalman3[2,0] <= 360)THEN
    x_kalman3[2,0] := x_kalman3[2,0]-360;
  END_IF

  F_kalman3[0,0]:=1;F_kalman3[0,1]:=0;F_kalman3[0,2]:= -1* x_kalman1[0,0]*COS(x_kalman2[0,0]*PI/180)*PLC_CYCLE;
  F_kalman3[1,0]:=0;F_kalman3[1,1]:=1;F_kalman3[1,2]:= -1* x_kalman1[0,0]*SIN(x_kalman2[0,0]*PI/180)*PLC_CYCLE;
  F_kalman3[2,0]:=0;F_kalman3[2,1]:=0;F_kalman3[2,2]:=1;
  //P_kalman3 = Fk_kalman3*P_kalman3*Fk_kalman3'+Q_kalman3;
    mulmat(F_kalman3,P_kalman3,tmp0,3,3,3);
    transpose(F_kalman3,Ft,3,3);   
    mulmat(tmp0,Ft,P_kalman3,3,3,3);
    accum(P_kalman3,Q_kalman3,3,3);

    setIdealAngle();

    robotAngle := x_kalman3[2,0];
    PosFdbckX :=  x_kalman3[0,0];
    PosFdbckY :=  x_kalman3[1,0];

END_FUNCTION_BLOCK

// ---- POUs/kalman/localization.TcPOU
FUNCTION_BLOCK localization
VAR_INPUT
END_VAR
VAR_OUTPUT
END_VAR
VAR
	rightMtrFdbck,leftMtrFdbck:LREAL;
END_VAR

 rightWheelFdbck:=-1 * robotdata.Position_Velocity.Locomotion_2_actual_velocity/reducer_ratio;
  leftWheelFdbck := robotdata.Position_Velocity.Locomotion_1_actual_velocity/reducer_ratio;
  linSpdFdbckRobot := (rightWheelFdbck+leftWheelFdbck)*2*PI/60*wheel_radius/2;
  angPosFdbckRobot := angPosFdbckRobot + (angSpdFdbckRobot+angSpdFdbckRobot_)/2*PLC_CYCLE;
  angPosFdbckRobot := angPosFdbckRobot + (angSpdFdbckRobot+angSpdFdbckRobot_)/2*PLC_CYCLE;
  angPosFdbckRobot_Abs:=angPosFdbckRobot_Abs + (angSpdFdbckRobot+angSpdFdbckRobot_)/2*PLC_CYCLE;
  angSpdFdbckRobot_ := angSpdFdbckRobot;
    
  angPosFdbckRobot:= myfmod(angPosFdbckRobot,360);

END_FUNCTION_BLOCK

// ---- POUs/kalman/cholsl.TcPOU
FUNCTION cholsl : INT
VAR_IN_OUT
	A:ARRAY[*,*] OF LREAL;
	aa:ARRAY[*,*] OF LREAL;
	p:ARRAY[*] OF LREAL;

END_VAR
VAR_INPUT
		n:SINT;
END_VAR
VAR
 i,j,k:SINT;
 sum:LREAL;
END_VAR

 IF (choldcsl((A),(aa),(p),n)=1) THEN
	cholsl:= 1;
	 return;
END_IF
    FOR i := 0 TO n-1 DO
        FOR j := i + 1  TO n-1 DO 
            aa[i,j] := 0.0;
        END_FOR
    END_FOR
	
    FOR i := 0 TO n-1 DO 
        aa[i,i] := aa[i,i] *aa[i,i];
        FOR k := i + 1 TO n-1 DO 
            aa[i,i] :=  aa[i,i] + aa[k,i] * aa[k,i];
		END_FOR
        FOR j := i + 1 TO n-1 DO 
            FOR k := j TO  n-1 DO
                aa[i,j] := aa[i,j]+ aa[k,i] * aa[k,j];
            END_FOR
        END_FOR
    END_FOR
    FOR i := 0 TO n-1 DO
        FOR j := 0 TO i-1 DO
            aa[i,j] := aa[j,i];
        END_FOR
    END_FOR

    cholsl:= 0;

END_FUNCTION

// ---- POUs/kalman/choldcsl.TcPOU
FUNCTION choldcsl : INT
VAR_IN_OUT
	A:ARRAY[*,*] OF LREAL;
	aa:ARRAY[*,*] OF LREAL;
	p:ARRAY[*] OF LREAL;
END_VAR
VAR_INPUT
		n:SINT;
END_VAR
VAR
 i,j,k:INT;
 sum:LREAL;

END_VAR


FOR i := 0 TO n-1 DO
	FOR j := 0 TO n-1 DO 
    	aa[i,j] := A[i,j];
		END_FOR
END_FOR
    	IF (choldc1(aa, p, n)=1) THEN
	 		choldcsl:=1;
			 return;
		END_IF

 
FOR i := 0 TO n-1 DO
         aa[i,i] := 1 / p[i];
        FOR j := i + 1 TO n-1 DO 
            sum := 0;
            FOR k := i TO j-1 DO 
                sum := sum-(aa[j,k] * aa[k,i]);
            END_FOR
            aa[j,i] := sum / p[j];
        END_FOR
END_FOR

    choldcsl:= 0;

END_FUNCTION

// ---- POUs/kalman/choldc1.TcPOU
FUNCTION choldc1 : INT
VAR_IN_OUT
	a:ARRAY[*,*] OF LREAL;
	p:ARRAY[*] OF LREAL;
	
END_VAR
VAR_INPUT
	n:SINT;
END_VAR
VAR
	i,j,k:INT;
 	sum:LREAL;
END_VAR

FOR i := 0 TO n-1 DO
            FOR j := i TO n-1 DO
              sum := a[i,j];
              FOR k := i - 1 TO 0 BY -1 DO
                sum := sum - (a[i,k] * a[j,k]);
	      	  END_FOR
              IF (i = j) THEN
                IF (sum <= 0) THEN
                  choldc1:=1;
				  return;
				  END_IF
		
                p[i] := SQRT(sum);
	     
              ELSE 
                a[j,i] := sum / p[i];
	      END_IF
	    END_FOR
	  END_FOR
    choldc1:=0;

END_FUNCTION

// ---- POUs/kalman/ssub.TcPOU
FUNCTION ssub : BOOL
VAR_IN_OUT
	a,b,c:ARRAY[*,*] OF LREAL;
END_VAR
VAR_INPUT
	n:SINT;
END_VAR
VAR
	j:SINT;
END_VAR

FOR j:=0 TO n-1 DO 
        c[0,j] := a[0,j] - b[0,j];
	END_FOR
	ssub:=true;

END_FUNCTION

// ---- POUs/kalman/sub_mat.TcPOU
FUNCTION sub_mat : BOOL
VAR_IN_OUT
	a:ARRAY[*,*] OF LREAL;
	b:ARRAY[*,*] OF LREAL;
	c:ARRAY[*,*] OF LREAL;


END_VAR
VAR_INPUT
		m,n:SINT;
END_VAR
VAR_OUTPUT
END_VAR
VAR
	i,j:int;
END_VAR

    FOR i:=0 TO m-1 DO
        FOR j:=0 TO n-1 DO
            c[i,j] := a[i,j]-b[i,j];
			END_FOR
			END_FOR
			sub_mat:=true;

END_FUNCTION

// ---- POUs/kalman/errorDegreeCalculator.TcPOU
FUNCTION errorDegreeCalculator : LREAL
VAR_INPUT
	in1,in2:LREAL;
END_VAR
VAR
	in1BigMapped,in2BigMapped,angPosDiff:LREAL;
END_VAR

 IF (in1BigMapped > 180) THEN
	in1BigMapped := in1BigMapped - 360;
	END_IF
  IF (in2BigMapped > 180) THEN
	in2BigMapped := in2BigMapped - 360;
	END_IF
  angPosDiff := in1BigMapped - in2BigMapped;
  IF (ABS(angPosDiff) > 180) THEN  
	errorDegreeCalculator:= angPosDiff - (mySign(angPosDiff) * 360);
  ELSE 
	errorDegreeCalculator:= angPosDiff;
	end_if

END_FUNCTION

// ---- POUs/kalman/mySign.TcPOU
FUNCTION mySign : int
VAR_INPUT
	 a:LREAL;
END_VAR
VAR
END_VAR

	IF (a < 0) THEN mySign:= -1;
    ELSIF (a>0) THEN mySign:= 1;
    ELSE mySign:= 0;
	
	END_IF

END_FUNCTION

// ---- POUs/kalman/setIdealAngle.TcPOU
FUNCTION setIdealAngle:bool
VAR_INPUT
END_VAR
VAR_OUTPUT
END_VAR
VAR
END_VAR

  IF (missionCompleted=1 OR  readyFlag=1)THEN
   // IF(( x_kalman3[2,0] <= 20 AND x_kalman3[2,0] >= 0) OR ( x_kalman3[2,0]<0 AND x_kalman3[2,0] >= -20)) THEN idealAngle := 0;
    IF(( x_kalman3[2,0] >= 70 AND x_kalman3[2,0] <= 110) OR (( x_kalman3[2,0] >= -290 AND x_kalman3[2,0] <= -250))) THEN 
		idealAngle := 90;
		robotdata.robot_direction := 3;
    ELSIF(( x_kalman3[2,0] <= -70 AND x_kalman3[2,0] >= -110))THEN  
	idealAngle:= -90;
	robotdata.robot_direction := 1;
    ELSIF (( x_kalman3[2,0] >= 160 AND x_kalman3[2,0] <= 200) OR ( x_kalman3[2,0] < -160 AND x_kalman3[2,0] >= -200)) THEN  
	idealAngle := -180;
	robotdata.robot_direction := 2;
	ELSE
	idealAngle:=0;	
	robotdata.robot_direction := 0;
	END_IF
    IF (readyFlag=1) THEN 
		readyFlag := 0;
		
	END_IF
  END_IF
  stabilization_yaw_deg:=detectStabilizedAngle(current_yaw:=robotdata.qr_yaw*180/PI);
  setIdealAngle:=true;

END_FUNCTION

// ---- POUs/kalman/kalmanController.TcPOU
FUNCTION_BLOCK kalmanController
VAR_INPUT
END_VAR
VAR_OUTPUT
END_VAR
VAR
	 linSpdCommand,fwdMoveSpdCommand,angMoveSpdCommand,angFwdPosError,angMovePosError,angFwdPosCommand,linSpdCommandShaped,linMoveSpdCommand,angSpdCommand:LREAL;
	 missionCompletedAng,missionCompletedLin:INT;
	 fb_kinematicSolution:kinematicSolution;
	 fb_localization:localization;
	 FB_DRIVE_MOTORS:DriveMotors();
END_VAR

IF (robotdata.motion_status = MOTION_ONGOING OR robotdata.motion_status = MOTION_ANGLE) AND (robotdata.activecommand=COMMAND_X_CORR OR robotdata.activecommand=COMMAND_ANG_CORR) THEN
	FB_DRIVE_MOTORS();


ELSIF(robotdata.controller=1)THEN
    fb_localization();
    missionCompletedLin := linPosErrGenerator(idealAngle,xGoal,yGoal,PosFdbckX,PosFdbckY,modeEnable);
    linMoveSpdCommand:= linPosErr* LINPOS_Kp;
    linSpdCommand := linSpdCommandMixer(modeEnable,linMoveSpdCommand,linPosErr);
    linSpdCommandShaped := linSpdCommandLimiter(linSpdCommand);
    angFwdPosCommand := forwardMovement(PosFdbckX,PosFdbckY,idealAngle);
    angMovePosError := angErrorCalc(AngPosCommand,robotAngle);
    angFwdPosError := angErrorCalc(angFwdPosCommand,robotAngle);
    angMoveSpdCommand := angMovePosError * TURNANG_Kp;
    fwdMoveSpdCommand := angFwdPosError* TURNFWD_Kp;
    
    missionCompletedAng:=angSpdCommandMixer(angMovePosError,modeEnable,angMoveSpdCommand,fwdMoveSpdCommand,angSpdCommand);
    angSpdCommandLimiter(angSpdCommand);
    missionCompleted:=(missionCompletedAng OR missionCompletedLin);
    IF(missionCompleted=1) THEN
		robotdata.motion_status:=MOTION_ENDED;
	END_IF
 
    fb_kinematicSolution(linSpdCommandShaped:=linSpdCommandShaped,angSpdCommand:=angSpdCommandShaped);

    IF (missionCompleted=1) THEN
       
      robotdata.motion_status := MOTION_ENDED;
	  robotdata.activeState:=MOVE_ENDED;
	  robotdata.Position_Velocity.Locomotion_1_target_velocity:= 0;
	  robotdata.Position_Velocity.Locomotion_2_target_velocity:= 0;
	  ELSE
		robotdata.Position_Velocity.Locomotion_1_target_velocity := leftMotorSpeedCommand;
		robotdata.Position_Velocity.Locomotion_2_target_velocity:=-1*rightMotorSpeedCommand;
	 END_IF
  END_IF

END_FUNCTION_BLOCK

// ---- POUs/kalman/kinematicSolution.TcPOU
FUNCTION_BLOCK kinematicSolution
VAR_INPUT
	 linSpdCommandShaped, angSpdCommand:LREAL;
END_VAR
VAR_OUTPUT
END_VAR
VAR
	v_left_radsec,v_right_radsec:LREAL;
END_VAR

 v_right_radsec:=((2*linSpdCommandShaped)+((angSpdCommand*PI/180)*ROBOT_RADIUS*2))/(2*WHEEL_RADIUS);
 rightMotorSpeedCommand:=LREAL_TO_DINT(LREAL_TO_DINT(v_right_radsec*60/(2*PI)*reducer_ratio));
  //printf("%ld-%ld,",v_right_radsec*60/(2*M_PI),*rightmtrspdcommand_rpm);
  v_left_radsec:=((2*linSpdCommandShaped)-((angSpdCommand*PI/180)*ROBOT_RADIUS*2))/(2*wheel_radius);
  leftMotorSpeedCommand:=LREAL_TO_DINT(LREAL_TO_DINT(v_left_radsec*60/(2*PI)*reducer_ratio));

END_FUNCTION_BLOCK

// ---- POUs/kalman/linPosErrGenerator.TcPOU
FUNCTION linPosErrGenerator : INT
VAR_INPUT
	lookingAngle,xGoal,yGoal,posFdbckX,posFdbckY:LREAL;
modeEnable:INT;
END_VAR
VAR
END_VAR

IF (lookingAngle = 0) THEN
    linPosErr := xGoal-posFdbckX;  
  ELSIF (lookingAngle = 180 OR lookingAngle = -180) THEN
    linPosErr := (xGoal-posFdbckX)*(-1);  
  else
    linPosErr := (yGoal-posFdbckY)*mySign(lookingAngle);
	END_IF
  // linPosErr = fabs(linPosErr);
  IF (modeEnable = 4 OR  modeEnable = 5) THEN
      // if (sqrt( ((xGoal-posFdbckX)*(xGoal-posFdbckX))+ ((yGoal-posFdbckY)*(yGoal-posFdbckY)) ) < 0.015)
      IF(ABS(linPosErr) < 0.005) THEN
          linPosErrGenerator:= 1;
		  return;
		  END_IF
		  END_IF
  linPosErrGenerator:= 0 ;

END_FUNCTION

// ---- POUs/kalman/linSpdCommandMixer.TcPOU
FUNCTION linSpdCommandMixer : LREAL
VAR_INPUT
	modeEnable:INT;
    linMoveSpdCommand, linPosErr:LREAL;
END_VAR
VAR
END_VAR

IF(modeEnable=0) THEN
    linSpdCommandMixer:= 0;
	return;
 ELSIF(modeEnable=4  OR modeEnable = 5)THEN
    IF(ABS(linPosErr)<0.005) THEN
       linSpdCommandMixer:=  0;
	   RETURN;
    else
       linSpdCommandMixer:=linMoveSpdCommand;   
	   RETURN;
	END_IF 
  END_IF
  linSpdCommandMixer:=  0;

END_FUNCTION

// ---- POUs/kalman/linSpdCommandLimiter.TcPOU
FUNCTION linSpdCommandLimiter : LREAL
VAR_INPUT
	LinSpdCmdIn:LREAL;
END_VAR
VAR
	accOut,jerkCmd,accCmd,LinSpdCmdOut:LREAL;
END_VAR

LinSpdCmdOut := 0;
  IF (modeEnable = 4 OR modeEnable = 5) THEN
  
    accCmd := (LinSpdCmdIn - LinSpdFdbck) / PLC_CYCLE;
    jerkCmd := (accCmd - accFdbck) / PLC_CYCLE;

    IF (jerkCmd > LINJERKLIMIT) THEN
      jerkCmd := LINJERKLIMIT;
	END_IF
    IF (jerkCmd < -1 * LINJERKLIMIT)THEN
      jerkCmd := -1 * LINJERKLIMIT;
	END_IF
    accOut := accFdbck + jerkCmd * PLC_CYCLE;

    IF (accOut > LINSPDRATELIMIT) THEN
      accOut := LINSPDRATELIMIT;
	  END_IF

    IF (accOut < -1 * LINSPDRATELIMIT)THEN
      accOut := -1 * LINSPDRATELIMIT;
END_IF
    LinSpdCmdOut := LinSpdFdbck + accOut * PLC_CYCLE;

    if (LinSpdCmdOut > FORWARD_MAX_SPEED)
    THEN
      LinSpdCmdOut:= FORWARD_MAX_SPEED;
      accOut := 0;
    END_IF

    if (LinSpdCmdOut < -1 * FORWARD_MAX_SPEED)
    THEN
      LinSpdCmdOut := -1 * FORWARD_MAX_SPEED;
      accOut := 0;
    END_IF

    LinSpdFdbck := LinSpdCmdOut;
    accFdbck := accOut;
  END_IF

  linSpdCommandLimiter:= LinSpdCmdOut;

END_FUNCTION

// ---- POUs/kalman/forwardMovement.TcPOU
FUNCTION forwardMovement : LREAL
VAR_INPUT
	PosFdbckX,PosFdbckY,idealAngle:LREAL;
END_VAR
VAR
	x2,y2,angForwardPosCommand,dist:LREAL;
	rot:ARRAY[0..1]OF ARRAY[0..1]OF LREAL;
END_VAR

  dist:=0.7;

  rot[0][0]:=COS(idealAngle*PI/180);
  rot[0][1]:=-1*SIN(idealAngle*PI/180);
  rot[1][0]:=SIN(idealAngle*PI/180);
  rot[1][1]:=COS(idealAngle*PI/180);

  IF (idealAngle=0 OR idealAngle=180 OR idealAngle=-180)THEN // Horizontal Solution
    IF ( modeEnable = 5)THEN
      x2 := PosFdbckX - rot[0][0] * dist;
      y2 := LREAL_TO_INT(PosFdbckY) - rot[1][0]*dist;
    
    ELSE
      x2 := PosFdbckX + rot[0][0] * dist;
      y2 := LREAL_TO_INT(PosFdbckY)+rot[1][0]*dist;
    END_IF
  
  ELSE // Vertical Solution
    IF(modeEnable = 5)THEN
      x2 := LREAL_TO_INT(PosFdbckX)  - rot[0][0] *dist;
      y2 := PosFdbckY - rot[1][0]*dist;
    
    ELSE 
      x2 := LREAL_TO_INT(PosFdbckX) + rot[0][0] *dist;
      y2 := PosFdbckY+rot[1][0]*dist;
    END_IF
  END_IF

  angForwardPosCommand := ATAN2(y2-PosFdbckY, x2-PosFdbckX)*180/PI;


 IF(modeEnable = 5)THEN
    IF(idealAngle = 0 OR idealAngle = -90) THEN
      forwardMovement:= angForwardPosCommand - 180;
    else
      forwardMovement:= angForwardPosCommand + 180;
  END_IF
  else
    forwardMovement:=  angForwardPosCommand;
	END_IF

END_FUNCTION

// ---- POUs/kalman/atan2.TcPOU
FUNCTION atan2 : LREAL
VAR_INPUT
	y,x:lreal;
END_VAR
VAR
END_VAR

IF(x>0)THEN
	atan2:=ATAN(y/x);
ELSIF(x<0 AND y>=0)THEN
	atan2:=ATAN(y/x)+PI;
ELSIF(x<0 AND y<0)THEN
	atan2:=ATAN(y/x)-PI;
ELSIF(x=0 AND y>0)THEN
	atan2:=PI/2;
ELSIF(x=0 AND y<0)THEN
	atan2:=-1*PI/2;
END_IF

END_FUNCTION

// ---- POUs/kalman/angErrorCalc.TcPOU
FUNCTION angErrorCalc : LREAL
VAR_INPUT
	 angPosCommand, angPosFdbck:LREAL;
END_VAR
VAR
	angPosDiff:LREAL;
END_VAR

IF(angPosCommand>180) THEN
angPosCommand:=180;
  ELSIF(angPosCommand< -180)THEN
 angPosCommand:=-180;
 END_IF
  angPosDiff:=angPosCommand-angPosFdbck;
  IF(abs(angPosDiff)>180) THEN
    angErrorCalc:= angPosDiff-mySign(angPosDiff)*360;
	RETURN;
  END_IF
  angErrorCalc:= angPosDiff;

END_FUNCTION

// ---- POUs/kalman/angSpdCommandMixer.TcPOU
FUNCTION angSpdCommandMixer : int
VAR_INPUT
	 angMovePosError:LREAL;
modeEnable :INT;
angMoveSpdCommand:LREAL;
forwardMoveSpdCommand:LREAL;
 
END_VAR
VAR_IN_OUT
 angSpdCommand:LREAL;
END_VAR
VAR
	missionCompletedAng:INT;
END_VAR

 missionCompletedAng := 0;
  IF (modeEnable = 0) THEN
      angSpdCommand := 0;
  ELSIF (modeEnable = 4 OR modeEnable = 5) THEN
      angSpdCommand := forwardMoveSpdCommand;   
  ELSE 
      IF (ABS(angMovePosError) < 0.2)THEN
          missionCompletedAng := 1;
          angSpdCommand := 0;
      ELSE
        angSpdCommand := angMoveSpdCommand;
		END_IF
  END_IF

  IF (modeEnable = 4 OR modeEnable = 5)  THEN
    ANGSPDRATELIMIT := 8;
  else 
    ANGSPDRATELIMIT := 50;
END_IF
  angSpdCommandMixer:= missionCompletedAng;

END_FUNCTION

// ---- POUs/kalman/angSpdCommandLimiter.TcPOU
FUNCTION angSpdCommandLimiter : LREAL
VAR_INPUT
	angSpdCommand:LREAL;
END_VAR
VAR
angRate:lreal;
END_VAR

angRate := (angSpdCommand - angSpdCommandShaped)/PLC_CYCLE;

  IF (ANGSPDRATELIMIT < angRate)THEN
    angRate := ANGSPDRATELIMIT;
  END_IF

  IF (-1*ANGSPDRATELIMIT > angRate)THEN
    angRate := -1 * ANGSPDRATELIMIT;
  END_IF

angSpdCommandShaped := angSpdCommandShaped+angRate * PLC_CYCLE;

IF(angSpdCommandShaped >= 40) THEN
 angSpdCommandShaped := 40;
 END_IF
IF(angSpdCommandShaped <= -40) THEN
 angSpdCommandShaped:= -40;
 END_IF
 angSpdCommandLimiter:=0;

END_FUNCTION

// ---- POUs/constrain_angle.TcPOU
FUNCTION constrain_angle:LREAL
VAR_INPUT
	angle:LREAL;
END_VAR
VAR_OUTPUT
	newangle:LREAL;
END_VAR
VAR
	x:LREAL;

END_VAR

 IF (ABS(roundToTwoDecimalPlaces(val:=x)) = roundToTwoDecimalPlaces(val:=PI)) THEN
    newangle:=x;
  END_IF

  x := lmod(x + PI, 2 * PI);
  IF (x < 0) THEN
    x :=x+ 2 * PI;
 END_IF
  newangle:= x - PI;
  constrain_angle:=newangle;

END_FUNCTION

// ---- POUs/roundToTwoDecimalPlaces.TcPOU
FUNCTION roundToTwoDecimalPlaces:LREAL
VAR_INPUT
	val:LREAL;
END_VAR
VAR_OUTPUT
	rval:LREAL;
END_VAR
VAR
	value:LREAL;
END_VAR

  value := LREAL_TO_DINT(val * 100 + 0.5);
  rval:= value/100;
  roundToTwoDecimalPlaces:=rval;

END_FUNCTION

// ---- POUs/set_imu_odeometry.TcPOU
FUNCTION set_imu_odeometry : BOOL
VAR_INPUT
END_VAR
VAR
	rr,icc_x,icc_y,current_y_state,current_x_state:LREAL;
END_VAR

current_x_state := robotdata.imu_state.imu_x;
current_y_state := robotdata.imu_state.imu_y;
IF (robotdata.imu_state.gyro_z = 0) THEN 
	robotdata.imu_state.gyro_z := 0.0000000000001;
END_IF
			rr := robotdata.encoder_v / robotdata.imu_state.gyro_z;
			icc_x :=  robotdata.imu_state.imu_x - (rr * SIN(robotdata.imu_state.imu_euler)); //instantaneous center of curvature
			icc_y := robotdata.imu_state.imu_y + (rr * COS(robotdata.imu_state.imu_euler)); // --
			 IF(pf_valid=0)THEN
			robotdata.imu_state.imu_x := ((current_x_state - icc_x) * COS(robotdata.imu_state.gyro_z * robotdata.imu_state.timediff)) - (current_y_state - icc_y) * SIN(robotdata.imu_state.gyro_z * robotdata.imu_state.timediff) + icc_x;
			robotdata.imu_state.imu_y := ((current_x_state - icc_x) * SIN(robotdata.imu_state.gyro_z * robotdata.imu_state.timediff)) + (current_y_state - icc_y) * COS(robotdata.imu_state.gyro_z * robotdata.imu_state.timediff) + icc_y;
			END_IF
			IF (ABS(robotdata.imu_state.gyro_z * robotdata.imu_state.timediff) > 0.00001)  THEN
				robotdata.imu_state.imu_euler := robotdata.imu_state.imu_euler + ((robotdata.imu_state.euler_yaw - imu_euler_prev) * PI / 180);
				imu_euler_prev := robotdata.imu_state.euler_yaw;
				//imu_euler=fmod((imu_euler+hr_gyro_z * timediff)+(2*M_PI), 2*M_PI);
			END_IF
set_imu_odeometry:=TRUE;

END_FUNCTION
